LIN {X 0,Y 539.247,Z 614.547,A -85,B 0,C 180,E1 4148.067,E2 4148.067} C_VEL
LIN {X 0,Y 539.704,Z 596.852,A -85,B 0,C 180,E1 4151.322,E2 4151.322} C_VEL
LIN {X 0,Y 540.471,Z 575.476,A -85,B 0,C 180,E1 4153.979,E2 4153.979} C_VEL
LIN {X 0,Y 541.317,Z 550.513,A -85,B 0,C 180,E1 4156.103,E2 4156.103} C_VEL
LIN {X 0,Y 542.051,Z 521.445,A -85,B 0,C 180,E1 4157.733,E2 4157.733} C_VEL
LIN {X 0,Y 542.484,Z 497.198,A -85,B 0,C 180,E1 4158.573,E2 4158.573} C_VEL
LIN {X 0,Y 539.142,Z 489.589,A -85,B 0,C 180,E1 4158.86,E2 4158.86} C_VEL
LIN {X 0,Y 531.289,Z 479.104,A -85,B 0,C 180,E1 4159.277,E2 4159.277} C_VEL
LIN {X 0,Y 530.945,Z 477.682,A -85,B 0,C 180,E1 4159.309,E2 4159.309} C_VEL
LIN {X 0,Y 530.735,Z 476.03,A -85,B 0,C 180,E1 4159.457,E2 4159.457} C_VEL
LIN {X 0,Y 530.499,Z 476.03,A -85,B 0,C 180,E1 4165.344,E2 4165.344} C_VEL
LIN {X 0,Y 530.255,Z 476.03,A -85,B 0,C 180,E1 4171.059,E2 4171.059} C_VEL
LIN {X 0,Y 530.287,Z 476.03,A -85,B 0,C 180,E1 4176.919,E2 4176.919} C_VEL
LIN {X 0,Y 530.344,Z 476.03,A -85,B 0,C 180,E1 4183.243,E2 4183.243} C_VEL
LIN {X 0,Y 530.21,Z 476.03,A -85,B 0,C 180,E1 4188.943,E2 4188.943} C_VEL
LIN {X 0,Y 530.367,Z 476.503,A -85,B 0,C 180,E1 4195.274,E2 4195.274} C_VEL
LIN {X 0,Y 532.518,Z 481.45,A -85,B 0,C 180,E1 4195.82,E2 4195.82} C_VEL
LIN {X 0,Y 542.624,Z 503.518,A -85,B 0,C 180,E1 4196.884,E2 4196.884} C_VEL
LIN {X 0,Y 542.117,Z 551.678,A -85,B 0,C 180,E1 4197.799,E2 4197.799} C_VEL
LIN {X 0,Y 540.712,Z 589.964,A -85,B 0,C 180,E1 4199.149,E2 4199.149} C_VEL
LIN {X 0,Y 538.696,Z 626.732,A -85,B 0,C 180,E1 4201.093,E2 4201.093} C_VEL
LIN {X 0,Y 536.576,Z 662.272,A -85,B 0,C 180,E1 4203.713,E2 4203.713} C_VEL
LIN {X 0,Y 534.555,Z 694.095,A -85,B 0,C 180,E1 4206.848,E2 4206.848} C_VEL
LIN {X 0,Y 532.935,Z 722.17,A -85,B 0,C 180,E1 4210.498,E2 4210.498} C_VEL
LIN {X 0,Y 531.902,Z 745.31,A -85,B 0,C 180,E1 4214.522,E2 4214.522} C_VEL
LIN {X 0,Y 531.296,Z 763.002,A -85,B 0,C 180,E1 4218.819,E2 4218.819} C_VEL
LIN {X 0,Y 531.132,Z 773.548,A -85,B 0,C 180,E1 4222.629,E2 4222.629} C_VEL
LIN {X 0,Y 531.001,Z 779.923,A -85,B 0,C 180,E1 4226.73,E2 4226.73} C_VEL
LIN {X 0,Y 531.003,Z 781.5,A -85,B 0,C 180,E1 4230,E2 4230} C_VEL
LIN {X 0,Y 531.007,Z 779.437,A -85,B 0,C 180,E1 4233.737,E2 4233.737} C_VEL
LIN {X 0,Y 531.193,Z 773.549,A -85,B 0,C 180,E1 4237.369,E2 4237.369} C_VEL
LIN {X 0,Y 531.407,Z 761.9,A -85,B 0,C 180,E1 4241.504,E2 4241.504} C_VEL
LIN {X 0,Y 531.939,Z 744.256,A -85,B 0,C 180,E1 4245.688,E2 4245.688} C_VEL
LIN {X 0,Y 533.035,Z 720.739,A -85,B 0,C 180,E1 4249.713,E2 4249.713} C_VEL
LIN {X 0,Y 534.71,Z 692.275,A -85,B 0,C 180,E1 4253.355,E2 4253.355} C_VEL
LIN {X 0,Y 536.74,Z 659.787,A -85,B 0,C 180,E1 4256.497,E2 4256.497} C_VEL
LIN {X 0,Y 538.885,Z 624.595,A -85,B 0,C 180,E1 4259.036,E2 4259.036} C_VEL
LIN {X 0,Y 540.782,Z 587.023,A -85,B 0,C 180,E1 4260.98,E2 4260.98} C_VEL
LIN {X 0,Y 542.348,Z 549.13,A -85,B 0,C 180,E1 4262.256,E2 4262.256} C_VEL
LIN {X 0,Y 542.002,Z 501.739,A -85,B 0,C 180,E1 4263.186,E2 4263.186} C_VEL
LIN {X 0,Y 532.957,Z 482.108,A -85,B 0,C 180,E1 4264.227,E2 4264.227} C_VEL
LIN {X 0,Y 530.337,Z 476.813,A -85,B 0,C 180,E1 4265.348,E2 4265.348} C_VEL
LIN {X 0,Y 530.278,Z 476.03,A -85,B 0,C 180,E1 4271.05,E2 4271.05} C_VEL
LIN {X 0,Y 530.271,Z 476.03,A -85,B 0,C 180,E1 4276.749,E2 4276.749} C_VEL
LIN {X 0,Y 530.233,Z 476.03,A -85,B 0,C 180,E1 4283.16,E2 4283.16} C_VEL
LIN {X 0,Y 530.371,Z 476.03,A -85,B 0,C 180,E1 4289.084,E2 4289.084} C_VEL
LIN {X 0,Y 530.381,Z 476.03,A -85,B 0,C 180,E1 4294.65,E2 4294.65} C_VEL
LIN {X 0,Y 530.532,Z 476.03,A -85,B 0,C 180,E1 4300.356,E2 4300.356} C_VEL
LIN {X 0,Y 530.613,Z 476.03,A -85,B 0,C 180,E1 4305.976,E2 4305.976} C_VEL
LIN {X 0,Y 530.721,Z 476.03,A -85,B 0,C 180,E1 4311.802,E2 4311.802} C_VEL
LIN {X 0,Y 530.902,Z 476.03,A -85,B 0,C 180,E1 4316.733,E2 4316.733} C_VEL
LIN {X 0,Y 530.989,Z 476.03,A -85,B 0,C 180,E1 4321.636,E2 4321.636} C_VEL
LIN {X 0,Y 530.878,Z 476.03,A -85,B 0,C 180,E1 4326.553,E2 4326.553} C_VEL
LIN {X 0,Y 530.677,Z 476.03,A -85,B 0,C 180,E1 4331.522,E2 4331.522} C_VEL
LIN {X 0,Y 530.569,Z 476.03,A -85,B 0,C 180,E1 4336.583,E2 4336.583} C_VEL
LIN {X 0,Y 530.55,Z 476.03,A -85,B 0,C 180,E1 4341.778,E2 4341.778} C_VEL
LIN {X 0,Y 530.375,Z 476.03,A -85,B 0,C 180,E1 4347.75,E2 4347.75} C_VEL
LIN {X 0,Y 530.316,Z 476.03,A -85,B 0,C 180,E1 4354.108,E2 4354.108} C_VEL
LIN {X 0,Y 530.322,Z 476.03,A -85,B 0,C 180,E1 4359.568,E2 4359.568} C_VEL
LIN {X 0,Y 530.322,Z 476.03,A -85,B 0,C 180,E1 4365.542,E2 4365.542} C_VEL
LIN {X 0,Y 530.274,Z 476.03,A -85,B 0,C 180,E1 4371.085,E2 4371.085} C_VEL
LIN {X 0,Y 530.239,Z 476.03,A -85,B 0,C 180,E1 4377.143,E2 4377.143} C_VEL
LIN {X 0,Y 530.401,Z 476.03,A -85,B 0,C 180,E1 4382.823,E2 4382.823} C_VEL
LIN {X 0,Y 530.547,Z 476.03,A -85,B 0,C 180,E1 4388.223,E2 4388.223} C_VEL
LIN {X 0,Y 530.576,Z 476.22,A -85,B 0,C 180,E1 4393.809,E2 4393.809} C_VEL
LIN {X 0,Y 541.216,Z 505.792,A -85,B 0,C 180,E1 4395.529,E2 4395.529} C_VEL
LIN {X 0,Y 539.385,Z 544.707,A -85,B 0,C 180,E1 4397.332,E2 4397.332} C_VEL
LIN {X 0,Y 537.207,Z 582.328,A -85,B 0,C 180,E1 4399.854,E2 4399.854} C_VEL
LIN {X 0,Y 535.231,Z 613.725,A -85,B 0,C 180,E1 4402.687,E2 4402.687} C_VEL
LIN {X 0,Y 533.459,Z 642.916,A -85,B 0,C 180,E1 4406.135,E2 4406.135} C_VEL
LIN {X 0,Y 532.186,Z 667.585,A -85,B 0,C 180,E1 4410,E2 4410} C_VEL
LIN {X 0,Y 531.51,Z 686.382,A -85,B 0,C 180,E1 4413.974,E2 4413.974} C_VEL
LIN {X 0,Y 531.15,Z 700.214,A -85,B 0,C 180,E1 4418.195,E2 4418.195} C_VEL
LIN {X 0,Y 531.001,Z 708.396,A -85,B 0,C 180,E1 4422.349,E2 4422.349} C_VEL
LIN {X 0,Y 530.857,Z 711.428,A -85,B 0,C 180,E1 4426.572,E2 4426.572} C_VEL
LIN {X 0,Y 530.911,Z 709.233,A -85,B 0,C 180,E1 4430.885,E2 4430.885} C_VEL
LIN {X 0,Y 531.121,Z 702.653,A -85,B 0,C 180,E1 4434.71,E2 4434.71} C_VEL
LIN {X 0,Y 531.447,Z 690.039,A -85,B 0,C 180,E1 4438.969,E2 4438.969} C_VEL
LIN {X 0,Y 531.996,Z 672.502,A -85,B 0,C 180,E1 4442.987,E2 4442.987} C_VEL
LIN {X 0,Y 533.086,Z 649.768,A -85,B 0,C 180,E1 4446.803,E2 4446.803} C_VEL
LIN {X 0,Y 534.693,Z 622.228,A -85,B 0,C 180,E1 4450.316,E2 4450.316} C_VEL
LIN {X 0,Y 536.712,Z 590.06,A -85,B 0,C 180,E1 4453.425,E2 4453.425} C_VEL
LIN {X 0,Y 538.829,Z 554.61,A -85,B 0,C 180,E1 4455.99,E2 4455.99} C_VEL
LIN {X 0,Y 540.802,Z 517.426,A -85,B 0,C 180,E1 4457.916,E2 4457.916} C_VEL
LIN {X 0,Y 540.909,Z 503.739,A -85,B 0,C 180,E1 4458.49,E2 4458.49} C_VEL
LIN {X 0,Y 530.23,Z 476.03,A -85,B 0,C 180,E1 4460.193,E2 4460.193} C_VEL
LIN {X 0,Y 530.366,Z 476.03,A -85,B 0,C 180,E1 4465.885,E2 4465.885} C_VEL
LIN {X 0,Y 530.428,Z 476.03,A -85,B 0,C 180,E1 4470.969,E2 4470.969} C_VEL
LIN {X 0,Y 530.383,Z 476.03,A -85,B 0,C 180,E1 4476.442,E2 4476.442} C_VEL
LIN {X 0,Y 530.49,Z 476.03,A -85,B 0,C 180,E1 4480.472,E2 4480.472} C_VEL
LIN {X 0,Y 534.953,Z 498.482,A -85,B 0,C 180,E1 4481.097,E2 4481.097} C_VEL
LIN {X 0,Y 534.252,Z 528.929,A -85,B 0,C 180,E1 4482.261,E2 4482.261} C_VEL
LIN {X 0,Y 533.467,Z 557.152,A -85,B 0,C 180,E1 4484.039,E2 4484.039} C_VEL
LIN {X 0,Y 532.623,Z 580.694,A -85,B 0,C 180,E1 4486.225,E2 4486.225} C_VEL
LIN {X 0,Y 531.918,Z 601.175,A -85,B 0,C 180,E1 4488.969,E2 4488.969} C_VEL
LIN {X 0,Y 531.468,Z 615.613,A -85,B 0,C 180,E1 4491.809,E2 4491.809} C_VEL
LIN {X 0,Y 531.266,Z 626.066,A -85,B 0,C 180,E1 4495.093,E2 4495.093} C_VEL
LIN {X 0,Y 531.115,Z 631.004,A -85,B 0,C 180,E1 4498.364,E2 4498.364} C_VEL
LIN {X 0,Y 531.116,Z 630.95,A -85,B 0,C 180,E1 4501.631,E2 4501.631} C_VEL
LIN {X 0,Y 531.225,Z 625.96,A -85,B 0,C 180,E1 4504.902,E2 4504.902} C_VEL
LIN {X 0,Y 531.465,Z 615.454,A -85,B 0,C 180,E1 4508.186,E2 4508.186} C_VEL
LIN {X 0,Y 532.021,Z 599.451,A -85,B 0,C 180,E1 4511.268,E2 4511.268} C_VEL
LIN {X 0,Y 532.805,Z 578.439,A -85,B 0,C 180,E1 4513.975,E2 4513.975} C_VEL
LIN {X 0,Y 533.692,Z 553.508,A -85,B 0,C 180,E1 4516.17,E2 4516.17} C_VEL
LIN {X 0,Y 534.446,Z 524.927,A -85,B 0,C 180,E1 4517.834,E2 4517.834} C_VEL
LIN {X 0,Y 534.92,Z 493.957,A -85,B 0,C 180,E1 4518.888,E2 4518.888} C_VEL
LIN {X 0,Y 530.945,Z 477.682,A -85,B 0,C 180,E1 4519.309,E2 4519.309} C_VEL
LIN {X 0,Y 529.475,Z 473.72,A -85,B 0,C 180,E1 4519.704,E2 4519.704} C_VEL
LIN {X 0,Y 526.146,Z 472.639,A -85,B 0,C 180,E1 4520.776,E2 4520.776} C_VEL
LIN {X 0,Y 522.532,Z 476.03,A -85,B 0,C 180,E1 4522.997,E2 4522.997} C_VEL
LIN {X 0,Y 522.452,Z 476.03,A -85,B 0,C 180,E1 4527.621,E2 4527.621} C_VEL
LIN {X 0,Y 522.345,Z 476.03,A -85,B 0,C 180,E1 4533.413,E2 4533.413} C_VEL
LIN {X 0,Y 522.405,Z 476.03,A -85,B 0,C 180,E1 4539.609,E2 4539.609} C_VEL
LIN {X 0,Y 522.398,Z 476.03,A -85,B 0,C 180,E1 4545.923,E2 4545.923} C_VEL
LIN {X 0,Y 522.272,Z 476.03,A -85,B 0,C 180,E1 4551.504,E2 4551.504} C_VEL
LIN {X 0,Y 522.352,Z 476.148,A -85,B 0,C 180,E1 4554.345,E2 4554.345} C_VEL
LIN {X 0,Y 523.947,Z 480.754,A -85,B 0,C 180,E1 4554.74,E2 4554.74} C_VEL
LIN {X 0,Y 527.796,Z 488.345,A -85,B 0,C 180,E1 4555.583,E2 4555.583} C_VEL
LIN {X 0,Y 536.066,Z 506.88,A -85,B 0,C 180,E1 4556.479,E2 4556.479} C_VEL
LIN {X 0,Y 535.382,Z 552.945,A -85,B 0,C 180,E1 4557.382,E2 4557.382} C_VEL
LIN {X 0,Y 533.76,Z 592.103,A -85,B 0,C 180,E1 4558.805,E2 4558.805} C_VEL
LIN {X 0,Y 531.495,Z 629.464,A -85,B 0,C 180,E1 4560.849,E2 4560.849} C_VEL
LIN {X 0,Y 529.142,Z 664.928,A -85,B 0,C 180,E1 4563.556,E2 4563.556} C_VEL
LIN {X 0,Y 526.827,Z 697.28,A -85,B 0,C 180,E1 4566.864,E2 4566.864} C_VEL
LIN {X 0,Y 525.14,Z 724.953,A -85,B 0,C 180,E1 4570.635,E2 4570.635} C_VEL
LIN {X 0,Y 524.066,Z 746.308,A -85,B 0,C 180,E1 4574.499,E2 4574.499} C_VEL
LIN {X 0,Y 523.413,Z 763.04,A -85,B 0,C 180,E1 4578.66,E2 4578.66} C_VEL
LIN {X 0,Y 523.257,Z 773.548,A -85,B 0,C 180,E1 4582.518,E2 4582.518} C_VEL
LIN {X 0,Y 523.117,Z 779.926,A -85,B 0,C 180,E1 4586.681,E2 4586.681} C_VEL
LIN {X 0,Y 523.114,Z 781.5,A -85,B 0,C 180,E1 4590,E2 4590} C_VEL
LIN {X 0,Y 523.173,Z 779.927,A -85,B 0,C 180,E1 4593.318,E2 4593.318} C_VEL
LIN {X 0,Y 523.313,Z 773.549,A -85,B 0,C 180,E1 4597.481,E2 4597.481} C_VEL
LIN {X 0,Y 523.542,Z 761.899,A -85,B 0,C 180,E1 4601.68,E2 4601.68} C_VEL
LIN {X 0,Y 524.109,Z 744.255,A -85,B 0,C 180,E1 4605.929,E2 4605.929} C_VEL
LIN {X 0,Y 525.393,Z 720.741,A -85,B 0,C 180,E1 4610.012,E2 4610.012} C_VEL
LIN {X 0,Y 527.246,Z 692.279,A -85,B 0,C 180,E1 4613.706,E2 4613.706} C_VEL
LIN {X 0,Y 529.499,Z 659.852,A -85,B 0,C 180,E1 4616.882,E2 4616.882} C_VEL
LIN {X 0,Y 531.856,Z 624.968,A -85,B 0,C 180,E1 4619.432,E2 4619.432} C_VEL
LIN {X 0,Y 533.86,Z 588.816,A -85,B 0,C 180,E1 4621.344,E2 4621.344} C_VEL
LIN {X 0,Y 535.619,Z 550.484,A -85,B 0,C 180,E1 4622.675,E2 4622.675} C_VEL
LIN {X 0,Y 535.515,Z 504.687,A -85,B 0,C 180,E1 4623.595,E2 4623.595} C_VEL
LIN {X 0,Y 528.216,Z 489.449,A -85,B 0,C 180,E1 4624.37,E2 4624.37} C_VEL
LIN {X 0,Y 523.102,Z 479.252,A -85,B 0,C 180,E1 4625.869,E2 4625.869} C_VEL
LIN {X 0,Y 522.384,Z 476.03,A -85,B 0,C 180,E1 4626.259,E2 4626.259} C_VEL
LIN {X 0,Y 522.392,Z 476.03,A -85,B 0,C 180,E1 4631.808,E2 4631.808} C_VEL
LIN {X 0,Y 522.295,Z 476.03,A -85,B 0,C 180,E1 4638.19,E2 4638.19} C_VEL
LIN {X 0,Y 522.325,Z 476.03,A -85,B 0,C 180,E1 4644.572,E2 4644.572} C_VEL
LIN {X 0,Y 522.419,Z 476.03,A -85,B 0,C 180,E1 4650.487,E2 4650.487} C_VEL
LIN {X 0,Y 522.489,Z 476.03,A -85,B 0,C 180,E1 4656.069,E2 4656.069} C_VEL
LIN {X 0,Y 522.628,Z 476.03,A -85,B 0,C 180,E1 4661.421,E2 4661.421} C_VEL
LIN {X 0,Y 522.747,Z 476.03,A -85,B 0,C 180,E1 4666.605,E2 4666.605} C_VEL
LIN {X 0,Y 522.803,Z 476.03,A -85,B 0,C 180,E1 4671.677,E2 4671.677} C_VEL
LIN {X 0,Y 523.019,Z 476.03,A -85,B 0,C 180,E1 4676.684,E2 4676.684} C_VEL
LIN {X 0,Y 523.081,Z 476.03,A -85,B 0,C 180,E1 4681.661,E2 4681.661} C_VEL
LIN {X 0,Y 522.95,Z 476.03,A -85,B 0,C 180,E1 4686.653,E2 4686.653} C_VEL
LIN {X 0,Y 522.744,Z 476.03,A -85,B 0,C 180,E1 4691.7,E2 4691.7} C_VEL
LIN {X 0,Y 522.609,Z 476.03,A -85,B 0,C 180,E1 4697.044,E2 4697.044} C_VEL
LIN {X 0,Y 522.616,Z 476.03,A -85,B 0,C 180,E1 4702.126,E2 4702.126} C_VEL
LIN {X 0,Y 522.481,Z 476.03,A -85,B 0,C 180,E1 4707.625,E2 4707.625} C_VEL
LIN {X 0,Y 522.392,Z 476.03,A -85,B 0,C 180,E1 4713.415,E2 4713.415} C_VEL
LIN {X 0,Y 522.418,Z 476.03,A -85,B 0,C 180,E1 4719.615,E2 4719.615} C_VEL
LIN {X 0,Y 522.434,Z 476.03,A -85,B 0,C 180,E1 4725.928,E2 4725.928} C_VEL
LIN {X 0,Y 522.325,Z 476.03,A -85,B 0,C 180,E1 4731.505,E2 4731.505} C_VEL
LIN {X 0,Y 522.35,Z 476.03,A -85,B 0,C 180,E1 4737.203,E2 4737.203} C_VEL
LIN {X 0,Y 522.46,Z 476.03,A -85,B 0,C 180,E1 4742.375,E2 4742.375} C_VEL
LIN {X 0,Y 522.626,Z 476.03,A -85,B 0,C 180,E1 4747.981,E2 4747.981} C_VEL
LIN {X 0,Y 522.696,Z 476.803,A -85,B 0,C 180,E1 4753.259,E2 4753.259} C_VEL
LIN {X 0,Y 534.354,Z 507.589,A -85,B 0,C 180,E1 4755.154,E2 4755.154} C_VEL
LIN {X 0,Y 532.357,Z 545.544,A -85,B 0,C 180,E1 4756.953,E2 4756.953} C_VEL
LIN {X 0,Y 529.992,Z 582.961,A -85,B 0,C 180,E1 4759.507,E2 4759.507} C_VEL
LIN {X 0,Y 527.703,Z 615.542,A -85,B 0,C 180,E1 4762.518,E2 4762.518} C_VEL
LIN {X 0,Y 525.768,Z 644.778,A -85,B 0,C 180,E1 4766.078,E2 4766.078} C_VEL
LIN {X 0,Y 524.34,Z 670.089,A -85,B 0,C 180,E1 4770.207,E2 4770.207} C_VEL
LIN {X 0,Y 523.628,Z 687.734,A -85,B 0,C 180,E1 4774.137,E2 4774.137} C_VEL
LIN {X 0,Y 523.253,Z 700.899,A -85,B 0,C 180,E1 4778.319,E2 4778.319} C_VEL
LIN {X 0,Y 523.093,Z 708.707,A -85,B 0,C 180,E1 4782.539,E2 4782.539} C_VEL
LIN {X 0,Y 522.927,Z 711.481,A -85,B 0,C 180,E1 4786.831,E2 4786.831} C_VEL
LIN {X 0,Y 523.026,Z 708.899,A -85,B 0,C 180,E1 4791.215,E2 4791.215} C_VEL
LIN {X 0,Y 523.253,Z 701.922,A -85,B 0,C 180,E1 4795.145,E2 4795.145} C_VEL
LIN {X 0,Y 523.574,Z 690.879,A -85,B 0,C 180,E1 4798.923,E2 4798.923} C_VEL
LIN {X 0,Y 524.186,Z 673.115,A -85,B 0,C 180,E1 4803.107,E2 4803.107} C_VEL
LIN {X 0,Y 525.368,Z 650.852,A -85,B 0,C 180,E1 4806.945,E2 4806.945} C_VEL
LIN {X 0,Y 527.251,Z 622.144,A -85,B 0,C 180,E1 4810.677,E2 4810.677} C_VEL
LIN {X 0,Y 529.548,Z 589.152,A -85,B 0,C 180,E1 4813.893,E2 4813.893} C_VEL
LIN {X 0,Y 531.773,Z 555.053,A -85,B 0,C 180,E1 4816.384,E2 4816.384} C_VEL
LIN {X 0,Y 533.964,Z 517.89,A -85,B 0,C 180,E1 4818.335,E2 4818.335} C_VEL
LIN {X 0,Y 533.752,Z 505.658,A -85,B 0,C 180,E1 4818.881,E2 4818.881} C_VEL
LIN {X 0,Y 522.34,Z 476.03,A -85,B 0,C 180,E1 4820.756,E2 4820.756} C_VEL
LIN {X 0,Y 522.477,Z 476.03,A -85,B 0,C 180,E1 4827.184,E2 4827.184} C_VEL
LIN {X 0,Y 522.428,Z 476.03,A -85,B 0,C 180,E1 4832.372,E2 4832.372} C_VEL
LIN {X 0,Y 522.501,Z 476.03,A -85,B 0,C 180,E1 4838.019,E2 4838.019} C_VEL
LIN {X 0,Y 522.576,Z 476.03,A -85,B 0,C 180,E1 4840.209,E2 4840.209} C_VEL
LIN {X 0,Y 527.382,Z 499.062,A -85,B 0,C 180,E1 4840.851,E2 4840.851} C_VEL
LIN {X 0,Y 526.676,Z 530.113,A -85,B 0,C 180,E1 4842.051,E2 4842.051} C_VEL
LIN {X 0,Y 525.903,Z 557.692,A -85,B 0,C 180,E1 4843.803,E2 4843.803} C_VEL
LIN {X 0,Y 524.978,Z 581.471,A -85,B 0,C 180,E1 4846.021,E2 4846.021} C_VEL
LIN {X 0,Y 524.285,Z 600.962,A -85,B 0,C 180,E1 4848.615,E2 4848.615} C_VEL
LIN {X 0,Y 523.73,Z 616.718,A -85,B 0,C 180,E1 4851.687,E2 4851.687} C_VEL
LIN {X 0,Y 523.509,Z 627.272,A -85,B 0,C 180,E1 4855.02,E2 4855.02} C_VEL
LIN {X 0,Y 523.341,Z 632.303,A -85,B 0,C 180,E1 4858.34,E2 4858.34} C_VEL
LIN {X 0,Y 523.342,Z 632.302,A -85,B 0,C 180,E1 4861.655,E2 4861.655} C_VEL
LIN {X 0,Y 523.469,Z 627.295,A -85,B 0,C 180,E1 4864.975,E2 4864.975} C_VEL
LIN {X 0,Y 523.761,Z 616.75,A -85,B 0,C 180,E1 4868.308,E2 4868.308} C_VEL
LIN {X 0,Y 524.343,Z 600.908,A -85,B 0,C 180,E1 4871.392,E2 4871.392} C_VEL
LIN {X 0,Y 525.063,Z 581.371,A -85,B 0,C 180,E1 4873.972,E2 4873.972} C_VEL
LIN {X 0,Y 526.047,Z 557.177,A -85,B 0,C 180,E1 4876.187,E2 4876.187} C_VEL
LIN {X 0,Y 526.817,Z 529.535,A -85,B 0,C 180,E1 4877.885,E2 4877.885} C_VEL
LIN {X 0,Y 527.321,Z 499.757,A -85,B 0,C 180,E1 4878.989,E2 4878.989} C_VEL
LIN {X 0,Y 525.63,Z 488.068,A -85,B 0,C 180,E1 4879.303,E2 4879.303} C_VEL
LIN {X 0,Y 522.848,Z 476.03,A -85,B 0,C 180,E1 4879.598,E2 4879.598} C_VEL
LIN {X 0,Y 522.532,Z 476.03,A -85,B 0,C 180,E1 4882.997,E2 4882.997} C_VEL
LIN {X 0,Y 520.003,Z 476.03,A -85,B 0,C 180,E1 4884.405,E2 4884.405} C_VEL
LIN {X 0,Y 514.507,Z 476.03,A -85,B 0,C 180,E1 4886.76,E2 4886.76} C_VEL
LIN {X 0,Y 514.399,Z 476.03,A -85,B 0,C 180,E1 4891.988,E2 4891.988} C_VEL
LIN {X 0,Y 514.428,Z 476.03,A -85,B 0,C 180,E1 4898.17,E2 4898.17} C_VEL
LIN {X 0,Y 514.498,Z 476.03,A -85,B 0,C 180,E1 4902.631,E2 4902.631} C_VEL
LIN {X 0,Y 514.419,Z 476.03,A -85,B 0,C 180,E1 4907.392,E2 4907.392} C_VEL
LIN {X 0,Y 514.4,Z 476.03,A -85,B 0,C 180,E1 4913.853,E2 4913.853} C_VEL
LIN {X 0,Y 517.886,Z 485.516,A -85,B 0,C 180,E1 4914.534,E2 4914.534} C_VEL
LIN {X 0,Y 523.589,Z 495.553,A -85,B 0,C 180,E1 4915.385,E2 4915.385} C_VEL
LIN {X 0,Y 529.466,Z 509.691,A -85,B 0,C 180,E1 4916.049,E2 4916.049} C_VEL
LIN {X 0,Y 528.646,Z 554.89,A -85,B 0,C 180,E1 4916.975,E2 4916.975} C_VEL
LIN {X 0,Y 526.855,Z 593.492,A -85,B 0,C 180,E1 4918.418,E2 4918.418} C_VEL
LIN {X 0,Y 524.414,Z 630.403,A -85,B 0,C 180,E1 4920.482,E2 4920.482} C_VEL
LIN {X 0,Y 521.864,Z 664.934,A -85,B 0,C 180,E1 4923.158,E2 4923.158} C_VEL
LIN {X 0,Y 519.387,Z 697.28,A -85,B 0,C 180,E1 4926.513,E2 4926.513} C_VEL
LIN {X 0,Y 517.459,Z 724.954,A -85,B 0,C 180,E1 4930.336,E2 4930.336} C_VEL
LIN {X 0,Y 516.251,Z 746.309,A -85,B 0,C 180,E1 4934.258,E2 4934.258} C_VEL
LIN {X 0,Y 515.568,Z 761.895,A -85,B 0,C 180,E1 4938.136,E2 4938.136} C_VEL
LIN {X 0,Y 515.356,Z 773.547,A -85,B 0,C 180,E1 4942.402,E2 4942.402} C_VEL
LIN {X 0,Y 515.211,Z 779.929,A -85,B 0,C 180,E1 4946.63,E2 4946.63} C_VEL
LIN {X 0,Y 515.214,Z 781.5,A -85,B 0,C 180,E1 4950,E2 4950} C_VEL
LIN {X 0,Y 515.278,Z 779.929,A -85,B 0,C 180,E1 4953.369,E2 4953.369} C_VEL
LIN {X 0,Y 515.433,Z 773.548,A -85,B 0,C 180,E1 4957.596,E2 4957.596} C_VEL
LIN {X 0,Y 515.664,Z 761.898,A -85,B 0,C 180,E1 4961.861,E2 4961.861} C_VEL
LIN {X 0,Y 516.324,Z 744.255,A -85,B 0,C 180,E1 4966.176,E2 4966.176} C_VEL
LIN {X 0,Y 517.711,Z 720.74,A -85,B 0,C 180,E1 4970.322,E2 4970.322} C_VEL
LIN {X 0,Y 519.777,Z 692.283,A -85,B 0,C 180,E1 4974.068,E2 4974.068} C_VEL
LIN {X 0,Y 522.296,Z 659.85,A -85,B 0,C 180,E1 4977.283,E2 4977.283} C_VEL
LIN {X 0,Y 524.906,Z 624.406,A -85,B 0,C 180,E1 4979.898,E2 4979.898} C_VEL
LIN {X 0,Y 527.077,Z 588.718,A -85,B 0,C 180,E1 4981.798,E2 4981.798} C_VEL
LIN {X 0,Y 528.931,Z 551.593,A -85,B 0,C 180,E1 4983.109,E2 4983.109} C_VEL
LIN {X 0,Y 529.011,Z 507.316,A -85,B 0,C 180,E1 4984.022,E2 4984.022} C_VEL
LIN {X 0,Y 521.991,Z 492.878,A -85,B 0,C 180,E1 4984.867,E2 4984.867} C_VEL
LIN {X 0,Y 515.836,Z 481.711,A -85,B 0,C 180,E1 4986.121,E2 4986.121} C_VEL
LIN {X 0,Y 514.502,Z 476.03,A -85,B 0,C 180,E1 4986.634,E2 4986.634} C_VEL
LIN {X 0,Y 514.461,Z 476.03,A -85,B 0,C 180,E1 4992.635,E2 4992.635} C_VEL
LIN {X 0,Y 514.369,Z 476.03,A -85,B 0,C 180,E1 4997.395,E2 4997.395} C_VEL
LIN {X 0,Y 514.359,Z 476.03,A -85,B 0,C 180,E1 5002.636,E2 5002.636} C_VEL
LIN {X 0,Y 514.541,Z 476.03,A -85,B 0,C 180,E1 5008.58,E2 5008.58} C_VEL
LIN {X 0,Y 514.488,Z 476.03,A -85,B 0,C 180,E1 5013.809,E2 5013.809} C_VEL
LIN {X 0,Y 514.601,Z 476.03,A -85,B 0,C 180,E1 5019.329,E2 5019.329} C_VEL
LIN {X 0,Y 514.787,Z 476.03,A -85,B 0,C 180,E1 5024.654,E2 5024.654} C_VEL
LIN {X 0,Y 514.881,Z 476.03,A -85,B 0,C 180,E1 5029.841,E2 5029.841} C_VEL
LIN {X 0,Y 515.109,Z 476.03,A -85,B 0,C 180,E1 5036.633,E2 5036.633} C_VEL
LIN {X 0,Y 515.105,Z 476.03,A -85,B 0,C 180,E1 5041.98,E2 5041.98} C_VEL
LIN {X 0,Y 515.038,Z 476.03,A -85,B 0,C 180,E1 5046.755,E2 5046.755} C_VEL
LIN {X 0,Y 514.814,Z 476.03,A -85,B 0,C 180,E1 5051.883,E2 5051.883} C_VEL
LIN {X 0,Y 514.713,Z 476.03,A -85,B 0,C 180,E1 5057.109,E2 5057.109} C_VEL
LIN {X 0,Y 514.67,Z 476.03,A -85,B 0,C 180,E1 5062.487,E2 5062.487} C_VEL
LIN {X 0,Y 514.528,Z 476.03,A -85,B 0,C 180,E1 5068.089,E2 5068.089} C_VEL
LIN {X 0,Y 514.421,Z 476.03,A -85,B 0,C 180,E1 5074.5,E2 5074.5} C_VEL
LIN {X 0,Y 514.475,Z 476.03,A -85,B 0,C 180,E1 5080.351,E2 5080.351} C_VEL
LIN {X 0,Y 514.442,Z 476.03,A -85,B 0,C 180,E1 5085.06,E2 5085.06} C_VEL
LIN {X 0,Y 514.482,Z 476.03,A -85,B 0,C 180,E1 5089.922,E2 5089.922} C_VEL
LIN {X 0,Y 514.362,Z 476.03,A -85,B 0,C 180,E1 5095.993,E2 5095.993} C_VEL
LIN {X 0,Y 514.52,Z 476.03,A -85,B 0,C 180,E1 5101.984,E2 5101.984} C_VEL
LIN {X 0,Y 514.659,Z 476.03,A -85,B 0,C 180,E1 5107.514,E2 5107.514} C_VEL
LIN {X 0,Y 514.729,Z 476.03,A -85,B 0,C 180,E1 5112.619,E2 5112.619} C_VEL
LIN {X 0,Y 527.453,Z 510.421,A -85,B 0,C 180,E1 5114.809,E2 5114.809} C_VEL
LIN {X 0,Y 525.258,Z 548.077,A -85,B 0,C 180,E1 5116.667,E2 5116.667} C_VEL
LIN {X 0,Y 522.683,Z 584.879,A -85,B 0,C 180,E1 5119.253,E2 5119.253} C_VEL
LIN {X 0,Y 520.142,Z 617.442,A -85,B 0,C 180,E1 5122.353,E2 5122.353} C_VEL
LIN {X 0,Y 518.128,Z 645.137,A -85,B 0,C 180,E1 5125.811,E2 5125.811} C_VEL
LIN {X 0,Y 516.617,Z 669.282,A -85,B 0,C 180,E1 5129.79,E2 5129.79} C_VEL
LIN {X 0,Y 515.781,Z 687.701,A -85,B 0,C 180,E1 5133.93,E2 5133.93} C_VEL
LIN {X 0,Y 515.425,Z 700.468,A -85,B 0,C 180,E1 5138.021,E2 5138.021} C_VEL
LIN {X 0,Y 515.221,Z 707.932,A -85,B 0,C 180,E1 5141.872,E2 5141.872} C_VEL
LIN {X 0,Y 515.018,Z 711.143,A -85,B 0,C 180,E1 5145.343,E2 5145.343} C_VEL
LIN {X 0,Y 515.026,Z 710.33,A -85,B 0,C 180,E1 5149.824,E2 5149.824} C_VEL
LIN {X 0,Y 515.299,Z 704.083,A -85,B 0,C 180,E1 5154.291,E2 5154.291} C_VEL
LIN {X 0,Y 515.695,Z 692.555,A -85,B 0,C 180,E1 5158.607,E2 5158.607} C_VEL
LIN {X 0,Y 516.323,Z 676.158,A -85,B 0,C 180,E1 5162.725,E2 5162.725} C_VEL
LIN {X 0,Y 517.603,Z 653.973,A -85,B 0,C 180,E1 5166.771,E2 5166.771} C_VEL
LIN {X 0,Y 519.535,Z 625.599,A -85,B 0,C 180,E1 5170.632,E2 5170.632} C_VEL
LIN {X 0,Y 521.893,Z 594.634,A -85,B 0,C 180,E1 5173.818,E2 5173.818} C_VEL
LIN {X 0,Y 524.516,Z 559.071,A -85,B 0,C 180,E1 5176.561,E2 5176.561} C_VEL
LIN {X 0,Y 526.915,Z 521.335,A -85,B 0,C 180,E1 5178.631,E2 5178.631} C_VEL
LIN {X 0,Y 527.1,Z 508.865,A -85,B 0,C 180,E1 5179.194,E2 5179.194} C_VEL
LIN {X 0,Y 514.411,Z 476.03,A -85,B 0,C 180,E1 5181.32,E2 5181.32} C_VEL
LIN {X 0,Y 514.555,Z 476.03,A -85,B 0,C 180,E1 5188.017,E2 5188.017} C_VEL
LIN {X 0,Y 514.488,Z 476.03,A -85,B 0,C 180,E1 5193.803,E2 5193.803} C_VEL
LIN {X 0,Y 514.629,Z 476.03,A -85,B 0,C 180,E1 5199.935,E2 5199.935} C_VEL
LIN {X 0,Y 519.755,Z 499.577,A -85,B 0,C 180,E1 5200.594,E2 5200.594} C_VEL
LIN {X 0,Y 519.156,Z 530.337,A -85,B 0,C 180,E1 5201.786,E2 5201.786} C_VEL
LIN {X 0,Y 518.332,Z 558.215,A -85,B 0,C 180,E1 5203.56,E2 5203.56} C_VEL
LIN {X 0,Y 517.319,Z 582.527,A -85,B 0,C 180,E1 5205.842,E2 5205.842} C_VEL
LIN {X 0,Y 516.561,Z 602.748,A -85,B 0,C 180,E1 5208.58,E2 5208.58} C_VEL
LIN {X 0,Y 515.981,Z 617.823,A -85,B 0,C 180,E1 5211.561,E2 5211.561} C_VEL
LIN {X 0,Y 515.735,Z 628.487,A -85,B 0,C 180,E1 5214.945,E2 5214.945} C_VEL
LIN {X 0,Y 515.556,Z 633.593,A -85,B 0,C 180,E1 5218.315,E2 5218.315} C_VEL
LIN {X 0,Y 515.582,Z 633.645,A -85,B 0,C 180,E1 5221.68,E2 5221.68} C_VEL
LIN {X 0,Y 515.734,Z 628.632,A -85,B 0,C 180,E1 5225.05,E2 5225.05} C_VEL
LIN {X 0,Y 516.061,Z 618.044,A -85,B 0,C 180,E1 5228.432,E2 5228.432} C_VEL
LIN {X 0,Y 516.711,Z 601.594,A -85,B 0,C 180,E1 5231.637,E2 5231.637} C_VEL
LIN {X 0,Y 517.601,Z 580.356,A -85,B 0,C 180,E1 5234.394,E2 5234.394} C_VEL
LIN {X 0,Y 518.575,Z 554.86,A -85,B 0,C 180,E1 5236.644,E2 5236.644} C_VEL
LIN {X 0,Y 519.329,Z 527.001,A -85,B 0,C 180,E1 5238.269,E2 5238.269} C_VEL
LIN {X 0,Y 519.745,Z 496.442,A -85,B 0,C 180,E1 5239.316,E2 5239.316} C_VEL
LIN {X 0,Y 514.907,Z 476.03,A -85,B 0,C 180,E1 5239.88,E2 5239.88} C_VEL
LIN {X 0,Y 514.588,Z 476.03,A -85,B 0,C 180,E1 5246.186,E2 5246.186} C_VEL
LIN {X 0,Y 514.507,Z 476.03,A -85,B 0,C 180,E1 5246.76,E2 5246.76} C_VEL
LIN {X 0,Y 510.554,Z 476.03,A -85,B 0,C 180,E1 5248.662,E2 5248.662} C_VEL
LIN {X 0,Y 506.494,Z 476.03,A -85,B 0,C 180,E1 5250.594,E2 5250.594} C_VEL
LIN {X 0,Y 506.514,Z 476.03,A -85,B 0,C 180,E1 5256.71,E2 5256.71} C_VEL
LIN {X 0,Y 506.509,Z 476.03,A -85,B 0,C 180,E1 5263.428,E2 5263.428} C_VEL
LIN {X 0,Y 506.416,Z 476.03,A -85,B 0,C 180,E1 5268.869,E2 5268.869} C_VEL
LIN {X 0,Y 506.47,Z 476.155,A -85,B 0,C 180,E1 5273.39,E2 5273.39} C_VEL
LIN {X 0,Y 512.056,Z 490.769,A -85,B 0,C 180,E1 5274.434,E2 5274.434} C_VEL
LIN {X 0,Y 519.906,Z 504.139,A -85,B 0,C 180,E1 5275.246,E2 5275.246} C_VEL
LIN {X 0,Y 522.752,Z 510.057,A -85,B 0,C 180,E1 5275.559,E2 5275.559} C_VEL
LIN {X 0,Y 522.001,Z 554.884,A -85,B 0,C 180,E1 5276.5,E2 5276.5} C_VEL
LIN {X 0,Y 520.033,Z 594.038,A -85,B 0,C 180,E1 5277.984,E2 5277.984} C_VEL
LIN {X 0,Y 517.419,Z 630.411,A -85,B 0,C 180,E1 5280.042,E2 5280.042} C_VEL
LIN {X 0,Y 514.538,Z 666.185,A -85,B 0,C 180,E1 5282.863,E2 5282.863} C_VEL
LIN {X 0,Y 511.843,Z 698.28,A -85,B 0,C 180,E1 5286.273,E2 5286.273} C_VEL
LIN {X 0,Y 509.782,Z 724.955,A -85,B 0,C 180,E1 5290.027,E2 5290.027} C_VEL
LIN {X 0,Y 508.427,Z 746.311,A -85,B 0,C 180,E1 5294.01,E2 5294.01} C_VEL
LIN {X 0,Y 507.704,Z 761.895,A -85,B 0,C 180,E1 5297.95,E2 5297.95} C_VEL
LIN {X 0,Y 507.456,Z 773.546,A -85,B 0,C 180,E1 5302.283,E2 5302.283} C_VEL
LIN {X 0,Y 507.306,Z 779.932,A -85,B 0,C 180,E1 5306.578,E2 5306.578} C_VEL
LIN {X 0,Y 507.327,Z 781.5,A -85,B 0,C 180,E1 5310,E2 5310} C_VEL
LIN {X 0,Y 507.371,Z 779.932,A -85,B 0,C 180,E1 5313.421,E2 5313.421} C_VEL
LIN {X 0,Y 507.526,Z 773.547,A -85,B 0,C 180,E1 5317.715,E2 5317.715} C_VEL
LIN {X 0,Y 507.818,Z 761.897,A -85,B 0,C 180,E1 5322.047,E2 5322.047} C_VEL
LIN {X 0,Y 508.55,Z 744.254,A -85,B 0,C 180,E1 5326.43,E2 5326.43} C_VEL
LIN {X 0,Y 510.001,Z 722.172,A -85,B 0,C 180,E1 5330.416,E2 5330.416} C_VEL
LIN {X 0,Y 512.182,Z 694.67,A -85,B 0,C 180,E1 5334.157,E2 5334.157} C_VEL
LIN {X 0,Y 514.879,Z 662.415,A -85,B 0,C 180,E1 5337.472,E2 5337.472} C_VEL
LIN {X 0,Y 517.645,Z 628.347,A -85,B 0,C 180,E1 5340.089,E2 5340.089} C_VEL
LIN {X 0,Y 520.096,Z 592.133,A -85,B 0,C 180,E1 5342.111,E2 5342.111} C_VEL
LIN {X 0,Y 522.19,Z 553.317,A -85,B 0,C 180,E1 5343.538,E2 5343.538} C_VEL
LIN {X 0,Y 522.564,Z 510.181,A -85,B 0,C 180,E1 5344.454,E2 5344.454} C_VEL
LIN {X 0,Y 515.365,Z 496.948,A -85,B 0,C 180,E1 5345.225,E2 5345.225} C_VEL
LIN {X 0,Y 509.297,Z 486.474,A -85,B 0,C 180,E1 5346.148,E2 5346.148} C_VEL
LIN {X 0,Y 506.532,Z 476.03,A -85,B 0,C 180,E1 5347.134,E2 5347.134} C_VEL
LIN {X 0,Y 506.473,Z 476.03,A -85,B 0,C 180,E1 5353.439,E2 5353.439} C_VEL
LIN {X 0,Y 506.388,Z 476.03,A -85,B 0,C 180,E1 5358.874,E2 5358.874} C_VEL
LIN {X 0,Y 506.511,Z 476.03,A -85,B 0,C 180,E1 5365.397,E2 5365.397} C_VEL
LIN {X 0,Y 506.508,Z 476.03,A -85,B 0,C 180,E1 5371.431,E2 5371.431} C_VEL
LIN {X 0,Y 506.653,Z 476.03,A -85,B 0,C 180,E1 5377.883,E2 5377.883} C_VEL
LIN {X 0,Y 506.856,Z 476.03,A -85,B 0,C 180,E1 5382.925,E2 5382.925} C_VEL
LIN {X 0,Y 506.865,Z 476.03,A -85,B 0,C 180,E1 5387.934,E2 5387.934} C_VEL
LIN {X 0,Y 506.964,Z 476.03,A -85,B 0,C 180,E1 5393.142,E2 5393.142} C_VEL
LIN {X 0,Y 507.082,Z 476.03,A -85,B 0,C 180,E1 5398.292,E2 5398.292} C_VEL
LIN {X 0,Y 507.072,Z 476.03,A -85,B 0,C 180,E1 5403.426,E2 5403.426} C_VEL
LIN {X 0,Y 506.914,Z 476.03,A -85,B 0,C 180,E1 5408.591,E2 5408.591} C_VEL
LIN {X 0,Y 506.834,Z 476.03,A -85,B 0,C 180,E1 5413.829,E2 5413.829} C_VEL
LIN {X 0,Y 506.753,Z 476.03,A -85,B 0,C 180,E1 5419.189,E2 5419.189} C_VEL
LIN {X 0,Y 506.702,Z 476.03,A -85,B 0,C 180,E1 5424.731,E2 5424.731} C_VEL
LIN {X 0,Y 506.537,Z 476.03,A -85,B 0,C 180,E1 5430.542,E2 5430.542} C_VEL
LIN {X 0,Y 506.561,Z 476.03,A -85,B 0,C 180,E1 5436.713,E2 5436.713} C_VEL
LIN {X 0,Y 506.46,Z 476.03,A -85,B 0,C 180,E1 5443.441,E2 5443.441} C_VEL
LIN {X 0,Y 506.491,Z 476.03,A -85,B 0,C 180,E1 5448.878,E2 5448.878} C_VEL
LIN {X 0,Y 506.453,Z 476.03,A -85,B 0,C 180,E1 5455.387,E2 5455.387} C_VEL
LIN {X 0,Y 506.536,Z 476.03,A -85,B 0,C 180,E1 5461.428,E2 5461.428} C_VEL
LIN {X 0,Y 506.75,Z 476.03,A -85,B 0,C 180,E1 5467.854,E2 5467.854} C_VEL
LIN {X 0,Y 506.856,Z 476.047,A -85,B 0,C 180,E1 5472.057,E2 5472.057} C_VEL
LIN {X 0,Y 520.632,Z 512.413,A -85,B 0,C 180,E1 5474.423,E2 5474.423} C_VEL
LIN {X 0,Y 518.256,Z 548.878,A -85,B 0,C 180,E1 5476.269,E2 5476.269} C_VEL
LIN {X 0,Y 515.452,Z 585.529,A -85,B 0,C 180,E1 5478.886,E2 5478.886} C_VEL
LIN {X 0,Y 512.574,Z 619.574,A -85,B 0,C 180,E1 5482.209,E2 5482.209} C_VEL
LIN {X 0,Y 510.421,Z 646.9,A -85,B 0,C 180,E1 5485.747,E2 5485.747} C_VEL
LIN {X 0,Y 508.808,Z 670.623,A -85,B 0,C 180,E1 5489.787,E2 5489.787} C_VEL
LIN {X 0,Y 507.898,Z 688.669,A -85,B 0,C 180,E1 5493.992,E2 5493.992} C_VEL
LIN {X 0,Y 507.506,Z 701.123,A -85,B 0,C 180,E1 5498.147,E2 5498.147} C_VEL
LIN {X 0,Y 507.299,Z 708.298,A -85,B 0,C 180,E1 5502.06,E2 5502.06} C_VEL
LIN {X 0,Y 507.088,Z 711.213,A -85,B 0,C 180,E1 5505.589,E2 5505.589} C_VEL
LIN {X 0,Y 507.123,Z 710.807,A -85,B 0,C 180,E1 5509.174,E2 5509.174} C_VEL
LIN {X 0,Y 507.374,Z 705.306,A -85,B 0,C 180,E1 5513.758,E2 5513.758} C_VEL
LIN {X 0,Y 507.699,Z 694.981,A -85,B 0,C 180,E1 5518.016,E2 5518.016} C_VEL
LIN {X 0,Y 508.453,Z 678.689,A -85,B 0,C 180,E1 5522.413,E2 5522.413} C_VEL
LIN {X 0,Y 509.67,Z 657.748,A -85,B 0,C 180,E1 5526.453,E2 5526.453} C_VEL
LIN {X 0,Y 511.668,Z 631.034,A -85,B 0,C 180,E1 5530.336,E2 5530.336} C_VEL
LIN {X 0,Y 514.403,Z 598.192,A -85,B 0,C 180,E1 5533.905,E2 5533.905} C_VEL
LIN {X 0,Y 517.273,Z 562.305,A -85,B 0,C 180,E1 5536.779,E2 5536.779} C_VEL
LIN {X 0,Y 519.832,Z 525.802,A -85,B 0,C 180,E1 5538.886,E2 5538.886} C_VEL
LIN {X 0,Y 520.147,Z 511.123,A -85,B 0,C 180,E1 5539.579,E2 5539.579} C_VEL
LIN {X 0,Y 506.454,Z 476.03,A -85,B 0,C 180,E1 5541.949,E2 5541.949} C_VEL
LIN {X 0,Y 506.562,Z 476.03,A -85,B 0,C 180,E1 5547.451,E2 5547.451} C_VEL
LIN {X 0,Y 506.581,Z 476.03,A -85,B 0,C 180,E1 5553.724,E2 5553.724} C_VEL
LIN {X 0,Y 506.774,Z 476.683,A -85,B 0,C 180,E1 5559.661,E2 5559.661} C_VEL
LIN {X 0,Y 512.233,Z 500.492,A -85,B 0,C 180,E1 5560.346,E2 5560.346} C_VEL
LIN {X 0,Y 511.605,Z 531.165,A -85,B 0,C 180,E1 5561.546,E2 5561.546} C_VEL
LIN {X 0,Y 510.757,Z 558.736,A -85,B 0,C 180,E1 5563.309,E2 5563.309} C_VEL
LIN {X 0,Y 509.641,Z 584.042,A -85,B 0,C 180,E1 5565.712,E2 5565.712} C_VEL
LIN {X 0,Y 508.819,Z 604.584,A -85,B 0,C 180,E1 5568.553,E2 5568.553} C_VEL
LIN {X 0,Y 508.157,Z 620.609,A -85,B 0,C 180,E1 5571.861,E2 5571.861} C_VEL
LIN {X 0,Y 507.976,Z 629.699,A -85,B 0,C 180,E1 5574.867,E2 5574.867} C_VEL
LIN {X 0,Y 507.783,Z 634.886,A -85,B 0,C 180,E1 5578.289,E2 5578.289} C_VEL
LIN {X 0,Y 507.808,Z 634.986,A -85,B 0,C 180,E1 5581.706,E2 5581.706} C_VEL
LIN {X 0,Y 507.976,Z 629.978,A -85,B 0,C 180,E1 5585.127,E2 5585.127} C_VEL
LIN {X 0,Y 508.354,Z 619.335,A -85,B 0,C 180,E1 5588.561,E2 5588.561} C_VEL
LIN {X 0,Y 509.033,Z 603.761,A -85,B 0,C 180,E1 5591.656,E2 5591.656} C_VEL
LIN {X 0,Y 509.834,Z 584.167,A -85,B 0,C 180,E1 5594.304,E2 5594.304} C_VEL
LIN {X 0,Y 510.878,Z 559.905,A -85,B 0,C 180,E1 5596.57,E2 5596.57} C_VEL
LIN {X 0,Y 511.662,Z 532.136,A -85,B 0,C 180,E1 5598.307,E2 5598.307} C_VEL
LIN {X 0,Y 512.169,Z 501.597,A -85,B 0,C 180,E1 5599.445,E2 5599.445} C_VEL
LIN {X 0,Y 508.728,Z 483.598,A -85,B 0,C 180,E1 5599.921,E2 5599.921} C_VEL
LIN {X 0,Y 506.974,Z 476.03,A -85,B 0,C 180,E1 5600.145,E2 5600.145} C_VEL
LIN {X 0,Y 506.612,Z 476.03,A -85,B 0,C 180,E1 5606.741,E2 5606.741} C_VEL
LIN {X 0,Y 506.494,Z 476.03,A -85,B 0,C 180,E1 5610.594,E2 5610.594} C_VEL
LIN {X 0,Y 502.368,Z 476.03,A -85,B 0,C 180,E1 5612.532,E2 5612.532} C_VEL
LIN {X 0,Y 498.503,Z 476.03,A -85,B 0,C 180,E1 5614.501,E2 5614.501} C_VEL
LIN {X 0,Y 498.533,Z 476.03,A -85,B 0,C 180,E1 5620.598,E2 5620.598} C_VEL
LIN {X 0,Y 498.553,Z 476.03,A -85,B 0,C 180,E1 5626.785,E2 5626.785} C_VEL
LIN {X 0,Y 498.513,Z 476.03,A -85,B 0,C 180,E1 5632.892,E2 5632.892} C_VEL
LIN {X 0,Y 503.893,Z 491.226,A -85,B 0,C 180,E1 5633.809,E2 5633.809} C_VEL
LIN {X 0,Y 513.82,Z 507.75,A -85,B 0,C 180,E1 5634.848,E2 5634.848} C_VEL
LIN {X 0,Y 516.359,Z 513.608,A -85,B 0,C 180,E1 5635.133,E2 5635.133} C_VEL
LIN {X 0,Y 515.332,Z 556.576,A -85,B 0,C 180,E1 5636.065,E2 5636.065} C_VEL
LIN {X 0,Y 513.179,Z 595.58,A -85,B 0,C 180,E1 5637.588,E2 5637.588} C_VEL
LIN {X 0,Y 510.308,Z 632.106,A -85,B 0,C 180,E1 5639.708,E2 5639.708} C_VEL
LIN {X 0,Y 507.218,Z 667.388,A -85,B 0,C 180,E1 5642.56,E2 5642.56} C_VEL
LIN {X 0,Y 504.427,Z 698.413,A -85,B 0,C 180,E1 5645.92,E2 5645.92} C_VEL
LIN {X 0,Y 502.089,Z 725.734,A -85,B 0,C 180,E1 5649.841,E2 5649.841} C_VEL
LIN {X 0,Y 500.645,Z 746.312,A -85,B 0,C 180,E1 5653.754,E2 5653.754} C_VEL
LIN {X 0,Y 499.851,Z 761.894,A -85,B 0,C 180,E1 5657.758,E2 5657.758} C_VEL
LIN {X 0,Y 499.571,Z 773.545,A -85,B 0,C 180,E1 5662.161,E2 5662.161} C_VEL
LIN {X 0,Y 499.401,Z 779.935,A -85,B 0,C 180,E1 5666.523,E2 5666.523} C_VEL
LIN {X 0,Y 499.44,Z 781.5,A -85,B 0,C 180,E1 5670,E2 5670} C_VEL
LIN {X 0,Y 499.463,Z 779.935,A -85,B 0,C 180,E1 5673.476,E2 5673.476} C_VEL
LIN {X 0,Y 499.63,Z 773.546,A -85,B 0,C 180,E1 5677.838,E2 5677.838} C_VEL
LIN {X 0,Y 499.957,Z 761.896,A -85,B 0,C 180,E1 5682.239,E2 5682.239} C_VEL
LIN {X 0,Y 500.816,Z 744.253,A -85,B 0,C 180,E1 5686.691,E2 5686.691} C_VEL
LIN {X 0,Y 502.478,Z 720.956,A -85,B 0,C 180,E1 5690.932,E2 5690.932} C_VEL
LIN {X 0,Y 504.982,Z 692.291,A -85,B 0,C 180,E1 5694.82,E2 5694.82} C_VEL
LIN {X 0,Y 507.956,Z 659.844,A -85,B 0,C 180,E1 5698.121,E2 5698.121} C_VEL
LIN {X 0,Y 510.957,Z 624.879,A -85,B 0,C 180,E1 5700.768,E2 5700.768} C_VEL
LIN {X 0,Y 513.596,Z 588.614,A -85,B 0,C 180,E1 5702.74,E2 5702.74} C_VEL
LIN {X 0,Y 515.731,Z 551.215,A -85,B 0,C 180,E1 5704.081,E2 5704.081} C_VEL
LIN {X 0,Y 515.875,Z 512.391,A -85,B 0,C 180,E1 5704.928,E2 5704.928} C_VEL
LIN {X 0,Y 509.679,Z 501.657,A -85,B 0,C 180,E1 5705.597,E2 5705.597} C_VEL
LIN {X 0,Y 501.356,Z 486.802,A -85,B 0,C 180,E1 5706.584,E2 5706.584} C_VEL
LIN {X 0,Y 498.654,Z 476.03,A -85,B 0,C 180,E1 5707.629,E2 5707.629} C_VEL
LIN {X 0,Y 498.548,Z 476.03,A -85,B 0,C 180,E1 5714.308,E2 5714.308} C_VEL
LIN {X 0,Y 498.435,Z 476.03,A -85,B 0,C 180,E1 5720.37,E2 5720.37} C_VEL
LIN {X 0,Y 498.632,Z 476.03,A -85,B 0,C 180,E1 5726.873,E2 5726.873} C_VEL
LIN {X 0,Y 498.598,Z 476.03,A -85,B 0,C 180,E1 5732.907,E2 5732.907} C_VEL
LIN {X 0,Y 498.754,Z 476.03,A -85,B 0,C 180,E1 5738.64,E2 5738.64} C_VEL
LIN {X 0,Y 498.936,Z 476.03,A -85,B 0,C 180,E1 5744.154,E2 5744.154} C_VEL
LIN {X 0,Y 499.024,Z 476.03,A -85,B 0,C 180,E1 5749.514,E2 5749.514} C_VEL
LIN {X 0,Y 499.158,Z 476.03,A -85,B 0,C 180,E1 5754.782,E2 5754.782} C_VEL
LIN {X 0,Y 499.293,Z 476.03,A -85,B 0,C 180,E1 5760.003,E2 5760.003} C_VEL
LIN {X 0,Y 499.196,Z 476.03,A -85,B 0,C 180,E1 5765.223,E2 5765.223} C_VEL
LIN {X 0,Y 499.037,Z 476.03,A -85,B 0,C 180,E1 5770.491,E2 5770.491} C_VEL
LIN {X 0,Y 498.905,Z 476.03,A -85,B 0,C 180,E1 5775.853,E2 5775.853} C_VEL
LIN {X 0,Y 498.833,Z 476.03,A -85,B 0,C 180,E1 5781.362,E2 5781.362} C_VEL
LIN {X 0,Y 498.679,Z 476.03,A -85,B 0,C 180,E1 5787.094,E2 5787.094} C_VEL
LIN {X 0,Y 498.565,Z 476.03,A -85,B 0,C 180,E1 5793.138,E2 5793.138} C_VEL
LIN {X 0,Y 498.536,Z 476.03,A -85,B 0,C 180,E1 5799.628,E2 5799.628} C_VEL
LIN {X 0,Y 498.575,Z 476.03,A -85,B 0,C 180,E1 5805.695,E2 5805.695} C_VEL
LIN {X 0,Y 498.504,Z 476.03,A -85,B 0,C 180,E1 5812.157,E2 5812.157} C_VEL
LIN {X 0,Y 498.499,Z 476.03,A -85,B 0,C 180,E1 5818.26,E2 5818.26} C_VEL
LIN {X 0,Y 498.661,Z 476.03,A -85,B 0,C 180,E1 5822.906,E2 5822.906} C_VEL
LIN {X 0,Y 498.847,Z 476.03,A -85,B 0,C 180,E1 5828.64,E2 5828.64} C_VEL
LIN {X 0,Y 498.946,Z 476.313,A -85,B 0,C 180,E1 5831.453,E2 5831.453} C_VEL
LIN {X 0,Y 513.526,Z 513.704,A -85,B 0,C 180,E1 5833.974,E2 5833.974} C_VEL
LIN {X 0,Y 511.161,Z 551.351,A -85,B 0,C 180,E1 5835.965,E2 5835.965} C_VEL
LIN {X 0,Y 508.275,Z 586.161,A -85,B 0,C 180,E1 5838.509,E2 5838.509} C_VEL
LIN {X 0,Y 505.102,Z 620.691,A -85,B 0,C 180,E1 5841.947,E2 5841.947} C_VEL
LIN {X 0,Y 502.681,Z 648.671,A -85,B 0,C 180,E1 5845.682,E2 5845.682} C_VEL
LIN {X 0,Y 501.008,Z 671.943,A -85,B 0,C 180,E1 5849.784,E2 5849.784} C_VEL
LIN {X 0,Y 500.05,Z 689.103,A -85,B 0,C 180,E1 5853.907,E2 5853.907} C_VEL
LIN {X 0,Y 499.66,Z 700.725,A -85,B 0,C 180,E1 5857.838,E2 5857.838} C_VEL
LIN {X 0,Y 499.361,Z 708.61,A -85,B 0,C 180,E1 5862.254,E2 5862.254} C_VEL
LIN {X 0,Y 499.169,Z 711.274,A -85,B 0,C 180,E1 5865.843,E2 5865.843} C_VEL
LIN {X 0,Y 499.191,Z 710.329,A -85,B 0,C 180,E1 5869.906,E2 5869.906} C_VEL
LIN {X 0,Y 499.479,Z 705.247,A -85,B 0,C 180,E1 5873.9,E2 5873.9} C_VEL
LIN {X 0,Y 499.839,Z 695.023,A -85,B 0,C 180,E1 5878.179,E2 5878.179} C_VEL
LIN {X 0,Y 500.649,Z 678.338,A -85,B 0,C 180,E1 5882.742,E2 5882.742} C_VEL
LIN {X 0,Y 502.177,Z 655.83,A -85,B 0,C 180,E1 5887.087,E2 5887.087} C_VEL
LIN {X 0,Y 504.35,Z 629.417,A -85,B 0,C 180,E1 5890.901,E2 5890.901} C_VEL
LIN {X 0,Y 507.242,Z 597.905,A -85,B 0,C 180,E1 5894.345,E2 5894.345} C_VEL
LIN {X 0,Y 510.357,Z 561.528,A -85,B 0,C 180,E1 5897.284,E2 5897.284} C_VEL
LIN {X 0,Y 513.11,Z 525.364,A -85,B 0,C 180,E1 5899.377,E2 5899.377} C_VEL
LIN {X 0,Y 513.467,Z 514.192,A -85,B 0,C 180,E1 5899.92,E2 5899.92} C_VEL
LIN {X 0,Y 499.228,Z 479.227,A -85,B 0,C 180,E1 5902.322,E2 5902.322} C_VEL
LIN {X 0,Y 498.551,Z 476.03,A -85,B 0,C 180,E1 5902.502,E2 5902.502} C_VEL
LIN {X 0,Y 498.642,Z 476.03,A -85,B 0,C 180,E1 5908.922,E2 5908.922} C_VEL
LIN {X 0,Y 498.682,Z 476.03,A -85,B 0,C 180,E1 5915.627,E2 5915.627} C_VEL
LIN {X 0,Y 498.783,Z 476.03,A -85,B 0,C 180,E1 5919.315,E2 5919.315} C_VEL
LIN {X 0,Y 504.826,Z 502.983,A -85,B 0,C 180,E1 5920.144,E2 5920.144} C_VEL
LIN {X 0,Y 504.024,Z 533.407,A -85,B 0,C 180,E1 5921.374,E2 5921.374} C_VEL
LIN {X 0,Y 503.046,Z 561.966,A -85,B 0,C 180,E1 5923.271,E2 5923.271} C_VEL
LIN {X 0,Y 501.932,Z 586.515,A -85,B 0,C 180,E1 5925.69,E2 5925.69} C_VEL
LIN {X 0,Y 501.11,Z 605.797,A -85,B 0,C 180,E1 5928.418,E2 5928.418} C_VEL
LIN {X 0,Y 500.425,Z 621.709,A -85,B 0,C 180,E1 5931.735,E2 5931.735} C_VEL
LIN {X 0,Y 500.215,Z 630.91,A -85,B 0,C 180,E1 5934.788,E2 5934.788} C_VEL
LIN {X 0,Y 499.994,Z 636.184,A -85,B 0,C 180,E1 5938.262,E2 5938.262} C_VEL
LIN {X 0,Y 500.034,Z 636.326,A -85,B 0,C 180,E1 5941.732,E2 5941.732} C_VEL
LIN {X 0,Y 500.246,Z 631.318,A -85,B 0,C 180,E1 5945.207,E2 5945.207} C_VEL
LIN {X 0,Y 500.644,Z 620.619,A -85,B 0,C 180,E1 5948.694,E2 5948.694} C_VEL
LIN {X 0,Y 501.405,Z 604.403,A -85,B 0,C 180,E1 5951.918,E2 5951.918} C_VEL
LIN {X 0,Y 502.347,Z 583.592,A -85,B 0,C 180,E1 5954.693,E2 5954.693} C_VEL
LIN {X 0,Y 503.383,Z 559.055,A -85,B 0,C 180,E1 5956.937,E2 5956.937} C_VEL
LIN {X 0,Y 504.161,Z 531.408,A -85,B 0,C 180,E1 5958.623,E2 5958.623} C_VEL
LIN {X 0,Y 504.617,Z 501.695,A -85,B 0,C 180,E1 5959.703,E2 5959.703} C_VEL
LIN {X 0,Y 499.021,Z 476.03,A -85,B 0,C 180,E1 5960.419,E2 5960.419} C_VEL
LIN {X 0,Y 498.656,Z 476.03,A -85,B 0,C 180,E1 5967.089,E2 5967.089} C_VEL
LIN {X 0,Y 498.519,Z 476.03,A -85,B 0,C 180,E1 5973.135,E2 5973.135} C_VEL
LIN {X 0,Y 498.503,Z 476.03,A -85,B 0,C 180,E1 5974.501,E2 5974.501} C_VEL
LIN {X 0,Y 496.052,Z 476.03,A -85,B 0,C 180,E1 5975.983,E2 5975.983} C_VEL
LIN {X 0,Y 490.674,Z 476.03,A -85,B 0,C 180,E1 5978.206,E2 5978.206} C_VEL
LIN {X 0,Y 490.573,Z 476.03,A -85,B 0,C 180,E1 5978.463,E2 5978.463} C_VEL
LIN {X 0,Y 490.651,Z 476.03,A -85,B 0,C 180,E1 5984.784,E2 5984.784} C_VEL
LIN {X 0,Y 490.537,Z 476.03,A -85,B 0,C 180,E1 5990.494,E2 5990.494} C_VEL
LIN {X 0,Y 490.618,Z 476.694,A -85,B 0,C 180,E1 5992.427,E2 5992.427} C_VEL
LIN {X 0,Y 501.071,Z 500.382,A -85,B 0,C 180,E1 5993.739,E2 5993.739} C_VEL
LIN {X 0,Y 508.998,Z 514.099,A -85,B 0,C 180,E1 5994.589,E2 5994.589} C_VEL
LIN {X 0,Y 509.717,Z 527.501,A -85,B 0,C 180,E1 5994.889,E2 5994.889} C_VEL
LIN {X 0,Y 507.978,Z 569.382,A -85,B 0,C 180,E1 5996.009,E2 5996.009} C_VEL
LIN {X 0,Y 505.631,Z 605.978,A -85,B 0,C 180,E1 5997.638,E2 5997.638} C_VEL
LIN {X 0,Y 502.511,Z 641.607,A -85,B 0,C 180,E1 5999.938,E2 5999.938} C_VEL
LIN {X 0,Y 499.242,Z 675.567,A -85,B 0,C 180,E1 6002.94,E2 6002.94} C_VEL
LIN {X 0,Y 496.303,Z 705.697,A -85,B 0,C 180,E1 6006.491,E2 6006.491} C_VEL
LIN {X 0,Y 494.099,Z 731.541,A -85,B 0,C 180,E1 6010.531,E2 6010.531} C_VEL
LIN {X 0,Y 492.649,Z 752.43,A -85,B 0,C 180,E1 6014.938,E2 6014.938} C_VEL
LIN {X 0,Y 491.92,Z 767.224,A -85,B 0,C 180,E1 6019.357,E2 6019.357} C_VEL
LIN {X 0,Y 491.629,Z 776.708,A -85,B 0,C 180,E1 6023.812,E2 6023.812} C_VEL
LIN {X 0,Y 491.552,Z 781.109,A -85,B 0,C 180,E1 6028.235,E2 6028.235} C_VEL
LIN {X 0,Y 491.65,Z 781.109,A -85,B 0,C 180,E1 6031.764,E2 6031.764} C_VEL
LIN {X 0,Y 491.613,Z 776.709,A -85,B 0,C 180,E1 6036.188,E2 6036.188} C_VEL
LIN {X 0,Y 491.938,Z 767.227,A -85,B 0,C 180,E1 6040.642,E2 6040.642} C_VEL
LIN {X 0,Y 492.599,Z 752.529,A -85,B 0,C 180,E1 6045.039,E2 6045.039} C_VEL
LIN {X 0,Y 494.134,Z 731.684,A -85,B 0,C 180,E1 6049.441,E2 6049.441} C_VEL
LIN {X 0,Y 496.337,Z 705.642,A -85,B 0,C 180,E1 6053.515,E2 6053.515} C_VEL
LIN {X 0,Y 499.23,Z 675.573,A -85,B 0,C 180,E1 6057.06,E2 6057.06} C_VEL
LIN {X 0,Y 502.504,Z 641.616,A -85,B 0,C 180,E1 6060.062,E2 6060.062} C_VEL
LIN {X 0,Y 505.536,Z 604.883,A -85,B 0,C 180,E1 6062.436,E2 6062.436} C_VEL
LIN {X 0,Y 508.12,Z 566.481,A -85,B 0,C 180,E1 6064.1,E2 6064.1} C_VEL
LIN {X 0,Y 510.023,Z 522.909,A -85,B 0,C 180,E1 6065.2,E2 6065.2} C_VEL
LIN {X 0,Y 509.081,Z 514.47,A -85,B 0,C 180,E1 6065.428,E2 6065.428} C_VEL
LIN {X 0,Y 494.968,Z 489.647,A -85,B 0,C 180,E1 6067.038,E2 6067.038} C_VEL
LIN {X 0,Y 491.515,Z 479.409,A -85,B 0,C 180,E1 6067.736,E2 6067.736} C_VEL
LIN {X 0,Y 490.68,Z 476.03,A -85,B 0,C 180,E1 6068.108,E2 6068.108} C_VEL
LIN {X 0,Y 490.664,Z 476.03,A -85,B 0,C 180,E1 6072.756,E2 6072.756} C_VEL
LIN {X 0,Y 490.563,Z 476.03,A -85,B 0,C 180,E1 6077.796,E2 6077.796} C_VEL
LIN {X 0,Y 490.579,Z 476.03,A -85,B 0,C 180,E1 6084.103,E2 6084.103} C_VEL
LIN {X 0,Y 490.653,Z 476.03,A -85,B 0,C 180,E1 6090.418,E2 6090.418} C_VEL
LIN {X 0,Y 490.77,Z 476.03,A -85,B 0,C 180,E1 6096.359,E2 6096.359} C_VEL
LIN {X 0,Y 490.957,Z 476.03,A -85,B 0,C 180,E1 6102.948,E2 6102.948} C_VEL
LIN {X 0,Y 491.107,Z 476.03,A -85,B 0,C 180,E1 6109.343,E2 6109.343} C_VEL
LIN {X 0,Y 491.242,Z 476.03,A -85,B 0,C 180,E1 6114.698,E2 6114.698} C_VEL
LIN {X 0,Y 491.392,Z 476.03,A -85,B 0,C 180,E1 6120.003,E2 6120.003} C_VEL
LIN {X 0,Y 491.285,Z 476.03,A -85,B 0,C 180,E1 6125.307,E2 6125.307} C_VEL
LIN {X 0,Y 491.119,Z 476.03,A -85,B 0,C 180,E1 6130.662,E2 6130.662} C_VEL
LIN {X 0,Y 490.943,Z 476.03,A -85,B 0,C 180,E1 6137.047,E2 6137.047} C_VEL
LIN {X 0,Y 490.871,Z 476.03,A -85,B 0,C 180,E1 6143.641,E2 6143.641} C_VEL
LIN {X 0,Y 490.639,Z 476.03,A -85,B 0,C 180,E1 6150.222,E2 6150.222} C_VEL
LIN {X 0,Y 490.607,Z 476.03,A -85,B 0,C 180,E1 6156.639,E2 6156.639} C_VEL
LIN {X 0,Y 490.625,Z 476.03,A -85,B 0,C 180,E1 6162.761,E2 6162.761} C_VEL
LIN {X 0,Y 490.683,Z 476.03,A -85,B 0,C 180,E1 6167.78,E2 6167.78} C_VEL
LIN {X 0,Y 490.558,Z 476.03,A -85,B 0,C 180,E1 6174.096,E2 6174.096} C_VEL
LIN {X 0,Y 490.626,Z 476.03,A -85,B 0,C 180,E1 6180.411,E2 6180.411} C_VEL
LIN {X 0,Y 490.858,Z 476.03,A -85,B 0,C 180,E1 6186.359,E2 6186.359} C_VEL
LIN {X 0,Y 490.996,Z 476.117,A -85,B 0,C 180,E1 6190.808,E2 6190.808} C_VEL
LIN {X 0,Y 505.654,Z 513.224,A -85,B 0,C 180,E1 6193.37,E2 6193.37} C_VEL
LIN {X 0,Y 506.734,Z 520.712,A -85,B 0,C 180,E1 6193.827,E2 6193.827} C_VEL
LIN {X 0,Y 503.714,Z 558.82,A -85,B 0,C 180,E1 6195.975,E2 6195.975} C_VEL
LIN {X 0,Y 500.304,Z 595.06,A -85,B 0,C 180,E1 6198.876,E2 6198.876} C_VEL
LIN {X 0,Y 497.273,Z 625.339,A -85,B 0,C 180,E1 6202.116,E2 6202.116} C_VEL
LIN {X 0,Y 494.709,Z 653.236,A -85,B 0,C 180,E1 6206.052,E2 6206.052} C_VEL
LIN {X 0,Y 492.934,Z 676.25,A -85,B 0,C 180,E1 6210.44,E2 6210.44} C_VEL
LIN {X 0,Y 492.093,Z 691.568,A -85,B 0,C 180,E1 6214.412,E2 6214.412} C_VEL
LIN {X 0,Y 491.651,Z 703.23,A -85,B 0,C 180,E1 6218.858,E2 6218.858} C_VEL
LIN {X 0,Y 491.442,Z 708.921,A -85,B 0,C 180,E1 6222.455,E2 6222.455} C_VEL
LIN {X 0,Y 491.207,Z 711.472,A -85,B 0,C 180,E1 6227.151,E2 6227.151} C_VEL
LIN {X 0,Y 491.4,Z 708.641,A -85,B 0,C 180,E1 6231.7,E2 6231.7} C_VEL
LIN {X 0,Y 491.72,Z 700.896,A -85,B 0,C 180,E1 6236.151,E2 6236.151} C_VEL
LIN {X 0,Y 492.33,Z 687.872,A -85,B 0,C 180,E1 6240.56,E2 6240.56} C_VEL
LIN {X 0,Y 493.443,Z 669.075,A -85,B 0,C 180,E1 6244.991,E2 6244.991} C_VEL
LIN {X 0,Y 495.565,Z 644.259,A -85,B 0,C 180,E1 6249.249,E2 6249.249} C_VEL
LIN {X 0,Y 498.352,Z 614.35,A -85,B 0,C 180,E1 6253.073,E2 6253.073} C_VEL
LIN {X 0,Y 501.494,Z 582.727,A -85,B 0,C 180,E1 6256.126,E2 6256.126} C_VEL
LIN {X 0,Y 504.784,Z 545.793,A -85,B 0,C 180,E1 6258.765,E2 6258.765} C_VEL
LIN {X 0,Y 506.724,Z 517.091,A -85,B 0,C 180,E1 6260.274,E2 6260.274} C_VEL
LIN {X 0,Y 492.236,Z 480.836,A -85,B 0,C 180,E1 6262.819,E2 6262.819} C_VEL
LIN {X 0,Y 490.58,Z 476.03,A -85,B 0,C 180,E1 6263.18,E2 6263.18} C_VEL
LIN {X 0,Y 490.756,Z 476.03,A -85,B 0,C 180,E1 6268.365,E2 6268.365} C_VEL
LIN {X 0,Y 490.716,Z 476.03,A -85,B 0,C 180,E1 6274.406,E2 6274.406} C_VEL
LIN {X 0,Y 490.878,Z 476.03,A -85,B 0,C 180,E1 6279.034,E2 6279.034} C_VEL
LIN {X 0,Y 497.318,Z 503.631,A -85,B 0,C 180,E1 6279.874,E2 6279.874} C_VEL
LIN {X 0,Y 496.472,Z 534.731,A -85,B 0,C 180,E1 6281.148,E2 6281.148} C_VEL
LIN {X 0,Y 495.418,Z 563.83,A -85,B 0,C 180,E1 6283.12,E2 6283.12} C_VEL
LIN {X 0,Y 494.24,Z 589,A -85,B 0,C 180,E1 6285.67,E2 6285.67} C_VEL
LIN {X 0,Y 493.334,Z 608.759,A -85,B 0,C 180,E1 6288.58,E2 6288.58} C_VEL
LIN {X 0,Y 492.673,Z 622.822,A -85,B 0,C 180,E1 6291.604,E2 6291.604} C_VEL
LIN {X 0,Y 492.456,Z 632.123,A -85,B 0,C 180,E1 6294.705,E2 6294.705} C_VEL
LIN {X 0,Y 492.216,Z 637.478,A -85,B 0,C 180,E1 6298.235,E2 6298.235} C_VEL
LIN {X 0,Y 492.283,Z 637.663,A -85,B 0,C 180,E1 6301.76,E2 6301.76} C_VEL
LIN {X 0,Y 492.489,Z 632.662,A -85,B 0,C 180,E1 6305.289,E2 6305.289} C_VEL
LIN {X 0,Y 492.94,Z 621.901,A -85,B 0,C 180,E1 6308.831,E2 6308.831} C_VEL
LIN {X 0,Y 493.737,Z 606.582,A -85,B 0,C 180,E1 6311.942,E2 6311.942} C_VEL
LIN {X 0,Y 494.694,Z 585.749,A -85,B 0,C 180,E1 6314.794,E2 6314.794} C_VEL
LIN {X 0,Y 495.791,Z 561.186,A -85,B 0,C 180,E1 6317.09,E2 6317.09} C_VEL
LIN {X 0,Y 496.608,Z 533.2,A -85,B 0,C 180,E1 6318.832,E2 6318.832} C_VEL
LIN {X 0,Y 497.087,Z 503.296,A -85,B 0,C 180,E1 6319.936,E2 6319.936} C_VEL
LIN {X 0,Y 491.107,Z 476.03,A -85,B 0,C 180,E1 6320.703,E2 6320.703} C_VEL
LIN {X 0,Y 490.712,Z 476.03,A -85,B 0,C 180,E1 6327.565,E2 6327.565} C_VEL
LIN {X 0,Y 490.6,Z 476.03,A -85,B 0,C 180,E1 6333.741,E2 6333.741} C_VEL
LIN {X 0,Y 490.573,Z 476.03,A -85,B 0,C 180,E1 6338.463,E2 6338.463} C_VEL
LIN {X 0,Y 488.014,Z 476.03,A -85,B 0,C 180,E1 6339.969,E2 6339.969} C_VEL
LIN {X 0,Y 482.684,Z 476.03,A -85,B 0,C 180,E1 6342.229,E2 6342.229} C_VEL
LIN {X 0,Y 482.595,Z 476.03,A -85,B 0,C 180,E1 6342.49,E2 6342.49} C_VEL
LIN {X 0,Y 482.62,Z 476.03,A -85,B 0,C 180,E1 6348.837,E2 6348.837} C_VEL
LIN {X 0,Y 482.67,Z 476.608,A -85,B 0,C 180,E1 6351.774,E2 6351.774} C_VEL
LIN {X 0,Y 496.031,Z 505.821,A -85,B 0,C 180,E1 6353.425,E2 6353.425} C_VEL
LIN {X 0,Y 503.232,Z 518.429,A -85,B 0,C 180,E1 6354.226,E2 6354.226} C_VEL
LIN {X 0,Y 501.534,Z 561.609,A -85,B 0,C 180,E1 6355.292,E2 6355.292} C_VEL
LIN {X 0,Y 499.045,Z 601.569,A -85,B 0,C 180,E1 6356.963,E2 6356.963} C_VEL
LIN {X 0,Y 496.157,Z 635.333,A -85,B 0,C 180,E1 6359.004,E2 6359.004} C_VEL
LIN {X 0,Y 492.631,Z 669.803,A -85,B 0,C 180,E1 6361.929,E2 6361.929} C_VEL
LIN {X 0,Y 489.504,Z 699.744,A -85,B 0,C 180,E1 6365.318,E2 6365.318} C_VEL
LIN {X 0,Y 486.765,Z 726.983,A -85,B 0,C 180,E1 6369.397,E2 6369.397} C_VEL
LIN {X 0,Y 485.033,Z 748.296,A -85,B 0,C 180,E1 6373.683,E2 6373.683} C_VEL
LIN {X 0,Y 484.117,Z 763.302,A -85,B 0,C 180,E1 6377.812,E2 6377.812} C_VEL
LIN {X 0,Y 483.803,Z 773.544,A -85,B 0,C 180,E1 6381.904,E2 6381.904} C_VEL
LIN {X 0,Y 483.598,Z 779.935,A -85,B 0,C 180,E1 6386.41,E2 6386.41} C_VEL
LIN {X 0,Y 483.656,Z 781.5,A -85,B 0,C 180,E1 6390,E2 6390} C_VEL
LIN {X 0,Y 483.673,Z 779.935,A -85,B 0,C 180,E1 6393.589,E2 6393.589} C_VEL
LIN {X 0,Y 483.844,Z 773.545,A -85,B 0,C 180,E1 6398.095,E2 6398.095} C_VEL
LIN {X 0,Y 484.254,Z 761.895,A -85,B 0,C 180,E1 6402.642,E2 6402.642} C_VEL
LIN {X 0,Y 485.292,Z 744.313,A -85,B 0,C 180,E1 6407.228,E2 6407.228} C_VEL
LIN {X 0,Y 487.232,Z 721.975,A -85,B 0,C 180,E1 6411.449,E2 6411.449} C_VEL
LIN {X 0,Y 489.98,Z 695.132,A -85,B 0,C 180,E1 6415.268,E2 6415.268} C_VEL
LIN {X 0,Y 493.359,Z 663.584,A -85,B 0,C 180,E1 6418.665,E2 6418.665} C_VEL
LIN {X 0,Y 496.831,Z 629.006,A -85,B 0,C 180,E1 6421.438,E2 6421.438} C_VEL
LIN {X 0,Y 499.754,Z 591.994,A -85,B 0,C 180,E1 6423.523,E2 6423.523} C_VEL
LIN {X 0,Y 502.308,Z 553.104,A -85,B 0,C 180,E1 6424.994,E2 6424.994} C_VEL
LIN {X 0,Y 503.093,Z 518.17,A -85,B 0,C 180,E1 6425.845,E2 6425.845} C_VEL
LIN {X 0,Y 489.668,Z 494.634,A -85,B 0,C 180,E1 6427.417,E2 6427.417} C_VEL
LIN {X 0,Y 482.965,Z 477.901,A -85,B 0,C 180,E1 6428.404,E2 6428.404} C_VEL
LIN {X 0,Y 482.729,Z 476.03,A -85,B 0,C 180,E1 6428.649,E2 6428.649} C_VEL
LIN {X 0,Y 482.665,Z 476.03,A -85,B 0,C 180,E1 6433.829,E2 6433.829} C_VEL
LIN {X 0,Y 482.604,Z 476.03,A -85,B 0,C 180,E1 6438.848,E2 6438.848} C_VEL
LIN {X 0,Y 482.684,Z 476.03,A -85,B 0,C 180,E1 6445.629,E2 6445.629} C_VEL
LIN {X 0,Y 482.707,Z 476.03,A -85,B 0,C 180,E1 6451.938,E2 6451.938} C_VEL
LIN {X 0,Y 482.885,Z 476.03,A -85,B 0,C 180,E1 6457.902,E2 6457.902} C_VEL
LIN {X 0,Y 483.071,Z 476.03,A -85,B 0,C 180,E1 6463.619,E2 6463.619} C_VEL
LIN {X 0,Y 483.179,Z 476.03,A -85,B 0,C 180,E1 6469.166,E2 6469.166} C_VEL
LIN {X 0,Y 483.341,Z 476.03,A -85,B 0,C 180,E1 6474.611,E2 6474.611} C_VEL
LIN {X 0,Y 483.522,Z 476.03,A -85,B 0,C 180,E1 6480.003,E2 6480.003} C_VEL
LIN {X 0,Y 483.385,Z 476.03,A -85,B 0,C 180,E1 6485.394,E2 6485.394} C_VEL
LIN {X 0,Y 483.189,Z 476.03,A -85,B 0,C 180,E1 6490.839,E2 6490.839} C_VEL
LIN {X 0,Y 483.048,Z 476.03,A -85,B 0,C 180,E1 6496.388,E2 6496.388} C_VEL
LIN {X 0,Y 482.971,Z 476.03,A -85,B 0,C 180,E1 6502.1,E2 6502.1} C_VEL
LIN {X 0,Y 482.759,Z 476.03,A -85,B 0,C 180,E1 6508.065,E2 6508.065} C_VEL
LIN {X 0,Y 482.663,Z 476.03,A -85,B 0,C 180,E1 6514.379,E2 6514.379} C_VEL
LIN {X 0,Y 482.691,Z 476.03,A -85,B 0,C 180,E1 6518.856,E2 6518.856} C_VEL
LIN {X 0,Y 482.661,Z 476.03,A -85,B 0,C 180,E1 6523.821,E2 6523.821} C_VEL
LIN {X 0,Y 482.69,Z 476.03,A -85,B 0,C 180,E1 6528.836,E2 6528.836} C_VEL
LIN {X 0,Y 482.608,Z 476.03,A -85,B 0,C 180,E1 6534.657,E2 6534.657} C_VEL
LIN {X 0,Y 482.711,Z 476.03,A -85,B 0,C 180,E1 6539.876,E2 6539.876} C_VEL
LIN {X 0,Y 482.896,Z 476.03,A -85,B 0,C 180,E1 6545.945,E2 6545.945} C_VEL
LIN {X 0,Y 483.061,Z 476.083,A -85,B 0,C 180,E1 6550.144,E2 6550.144} C_VEL
LIN {X 0,Y 497.562,Z 512.15,A -85,B 0,C 180,E1 6552.695,E2 6552.695} C_VEL
LIN {X 0,Y 500,Z 521.84,A -85,B 0,C 180,E1 6553.376,E2 6553.376} C_VEL
LIN {X 0,Y 496.9,Z 558.042,A -85,B 0,C 180,E1 6555.441,E2 6555.441} C_VEL
LIN {X 0,Y 493.202,Z 594.468,A -85,B 0,C 180,E1 6558.378,E2 6558.378} C_VEL
LIN {X 0,Y 489.937,Z 624.945,A -85,B 0,C 180,E1 6561.667,E2 6561.667} C_VEL
LIN {X 0,Y 487.1,Z 653.564,A -85,B 0,C 180,E1 6565.767,E2 6565.767} C_VEL
LIN {X 0,Y 485.134,Z 676.866,A -85,B 0,C 180,E1 6570.305,E2 6570.305} C_VEL
LIN {X 0,Y 484.21,Z 692.399,A -85,B 0,C 180,E1 6574.484,E2 6574.484} C_VEL
LIN {X 0,Y 483.771,Z 703.793,A -85,B 0,C 180,E1 6579.004,E2 6579.004} C_VEL
LIN {X 0,Y 483.502,Z 709.234,A -85,B 0,C 180,E1 6582.663,E2 6582.663} C_VEL
LIN {X 0,Y 483.345,Z 711.395,A -85,B 0,C 180,E1 6586.376,E2 6586.376} C_VEL
LIN {X 0,Y 483.399,Z 710.219,A -85,B 0,C 180,E1 6590.154,E2 6590.154} C_VEL
LIN {X 0,Y 483.748,Z 703.984,A -85,B 0,C 180,E1 6594.814,E2 6594.814} C_VEL
LIN {X 0,Y 484.284,Z 692.448,A -85,B 0,C 180,E1 6599.407,E2 6599.407} C_VEL
LIN {X 0,Y 485.186,Z 676.266,A -85,B 0,C 180,E1 6603.737,E2 6603.737} C_VEL
LIN {X 0,Y 487.084,Z 653.7,A -85,B 0,C 180,E1 6608.119,E2 6608.119} C_VEL
LIN {X 0,Y 489.918,Z 625.344,A -85,B 0,C 180,E1 6612.19,E2 6612.19} C_VEL
LIN {X 0,Y 493.104,Z 595.487,A -85,B 0,C 180,E1 6615.439,E2 6615.439} C_VEL
LIN {X 0,Y 496.676,Z 560.316,A -85,B 0,C 180,E1 6618.311,E2 6618.311} C_VEL
LIN {X 0,Y 499.819,Z 524.168,A -85,B 0,C 180,E1 6620.417,E2 6620.417} C_VEL
LIN {X 0,Y 499.506,Z 518.524,A -85,B 0,C 180,E1 6620.745,E2 6620.745} C_VEL
LIN {X 0,Y 485.04,Z 482.71,A -85,B 0,C 180,E1 6623.342,E2 6623.342} C_VEL
LIN {X 0,Y 482.7,Z 476.03,A -85,B 0,C 180,E1 6623.745,E2 6623.745} C_VEL
LIN {X 0,Y 482.784,Z 476.03,A -85,B 0,C 180,E1 6629.88,E2 6629.88} C_VEL
LIN {X 0,Y 482.803,Z 476.03,A -85,B 0,C 180,E1 6635.939,E2 6635.939} C_VEL
LIN {X 0,Y 482.979,Z 476.03,A -85,B 0,C 180,E1 6638.722,E2 6638.722} C_VEL
LIN {X 0,Y 489.75,Z 505.894,A -85,B 0,C 180,E1 6639.649,E2 6639.649} C_VEL
LIN {X 0,Y 488.931,Z 537.227,A -85,B 0,C 180,E1 6640.985,E2 6640.985} C_VEL
LIN {X 0,Y 487.821,Z 565.655,A -85,B 0,C 180,E1 6642.965,E2 6642.965} C_VEL
LIN {X 0,Y 486.587,Z 589.835,A -85,B 0,C 180,E1 6645.45,E2 6645.45} C_VEL
LIN {X 0,Y 485.623,Z 610.48,A -85,B 0,C 180,E1 6648.533,E2 6648.533} C_VEL
LIN {X 0,Y 484.865,Z 625.582,A -85,B 0,C 180,E1 6651.92,E2 6651.92} C_VEL
LIN {X 0,Y 484.571,Z 635.201,A -85,B 0,C 180,E1 6655.517,E2 6655.517} C_VEL
LIN {X 0,Y 484.451,Z 638.77,A -85,B 0,C 180,E1 6658.206,E2 6658.206} C_VEL
LIN {X 0,Y 484.521,Z 639.002,A -85,B 0,C 180,E1 6661.788,E2 6661.788} C_VEL
LIN {X 0,Y 484.759,Z 634.009,A -85,B 0,C 180,E1 6665.374,E2 6665.374} C_VEL
LIN {X 0,Y 485.235,Z 623.195,A -85,B 0,C 180,E1 6668.972,E2 6668.972} C_VEL
LIN {X 0,Y 486.087,Z 607.759,A -85,B 0,C 180,E1 6672.134,E2 6672.134} C_VEL
LIN {X 0,Y 487.106,Z 586.862,A -85,B 0,C 180,E1 6675.017,E2 6675.017} C_VEL
LIN {X 0,Y 488.27,Z 561.89,A -85,B 0,C 180,E1 6677.362,E2 6677.362} C_VEL
LIN {X 0,Y 489.123,Z 533.592,A -85,B 0,C 180,E1 6679.116,E2 6679.116} C_VEL
LIN {X 0,Y 489.59,Z 502.177,A -85,B 0,C 180,E1 6680.249,E2 6680.249} C_VEL
LIN {X 0,Y 483.141,Z 476.03,A -85,B 0,C 180,E1 6680.988,E2 6680.988} C_VEL
LIN {X 0,Y 482.871,Z 476.03,A -85,B 0,C 180,E1 6686.034,E2 6686.034} C_VEL
LIN {X 0,Y 482.677,Z 476.03,A -85,B 0,C 180,E1 6692.221,E2 6692.221} C_VEL
LIN {X 0,Y 482.672,Z 476.03,A -85,B 0,C 180,E1 6698.851,E2 6698.851} C_VEL
LIN {X 0,Y 482.595,Z 476.03,A -85,B 0,C 180,E1 6702.49,E2 6702.49} C_VEL
LIN {X 0,Y 480.059,Z 476.03,A -85,B 0,C 180,E1 6704.024,E2 6704.024} C_VEL
LIN {X 0,Y 474.705,Z 476.03,A -85,B 0,C 180,E1 6706.325,E2 6706.325} C_VEL
LIN {X 0,Y 474.618,Z 476.03,A -85,B 0,C 180,E1 6706.592,E2 6706.592} C_VEL
LIN {X 0,Y 474.728,Z 476.266,A -85,B 0,C 180,E1 6711.037,E2 6711.037} C_VEL
LIN {X 0,Y 490.637,Z 510.685,A -85,B 0,C 180,E1 6713.07,E2 6713.07} C_VEL
LIN {X 0,Y 496.505,Z 520.581,A -85,B 0,C 180,E1 6713.742,E2 6713.742} C_VEL
LIN {X 0,Y 494.536,Z 564.715,A -85,B 0,C 180,E1 6714.933,E2 6714.933} C_VEL
LIN {X 0,Y 491.579,Z 606.228,A -85,B 0,C 180,E1 6716.791,E2 6716.791} C_VEL
LIN {X 0,Y 488.157,Z 644.112,A -85,B 0,C 180,E1 6719.244,E2 6719.244} C_VEL
LIN {X 0,Y 485.071,Z 673.868,A -85,B 0,C 180,E1 6721.889,E2 6721.889} C_VEL
LIN {X 0,Y 481.422,Z 705.186,A -85,B 0,C 180,E1 6725.644,E2 6725.644} C_VEL
LIN {X 0,Y 478.745,Z 731.549,A -85,B 0,C 180,E1 6729.882,E2 6729.882} C_VEL
LIN {X 0,Y 477.059,Z 752.092,A -85,B 0,C 180,E1 6734.349,E2 6734.349} C_VEL
LIN {X 0,Y 476.148,Z 767.222,A -85,B 0,C 180,E1 6739,E2 6739} C_VEL
LIN {X 0,Y 475.838,Z 776.706,A -85,B 0,C 180,E1 6743.605,E2 6743.605} C_VEL
LIN {X 0,Y 475.742,Z 781.108,A -85,B 0,C 180,E1 6748.176,E2 6748.176} C_VEL
LIN {X 0,Y 475.853,Z 781.108,A -85,B 0,C 180,E1 6751.823,E2 6751.823} C_VEL
LIN {X 0,Y 475.83,Z 776.707,A -85,B 0,C 180,E1 6756.394,E2 6756.394} C_VEL
LIN {X 0,Y 476.229,Z 767.224,A -85,B 0,C 180,E1 6760.997,E2 6760.997} C_VEL
LIN {X 0,Y 477.025,Z 752.096,A -85,B 0,C 180,E1 6765.652,E2 6765.652} C_VEL
LIN {X 0,Y 478.796,Z 731.553,A -85,B 0,C 180,E1 6770.115,E2 6770.115} C_VEL
LIN {X 0,Y 481.446,Z 705.342,A -85,B 0,C 180,E1 6774.332,E2 6774.332} C_VEL
LIN {X 0,Y 484.86,Z 675.572,A -85,B 0,C 180,E1 6777.931,E2 6777.931} C_VEL
LIN {X 0,Y 488.182,Z 644.054,A -85,B 0,C 180,E1 6780.768,E2 6780.768} C_VEL
LIN {X 0,Y 491.589,Z 605.88,A -85,B 0,C 180,E1 6783.273,E2 6783.273} C_VEL
LIN {X 0,Y 494.795,Z 564.877,A -85,B 0,C 180,E1 6785.115,E2 6785.115} C_VEL
LIN {X 0,Y 497.048,Z 521.695,A -85,B 0,C 180,E1 6786.274,E2 6786.274} C_VEL
LIN {X 0,Y 484.083,Z 498.859,A -85,B 0,C 180,E1 6787.846,E2 6787.846} C_VEL
LIN {X 0,Y 474.779,Z 476.03,A -85,B 0,C 180,E1 6789.198,E2 6789.198} C_VEL
LIN {X 0,Y 474.648,Z 476.03,A -85,B 0,C 180,E1 6795.437,E2 6795.437} C_VEL
LIN {X 0,Y 474.614,Z 476.03,A -85,B 0,C 180,E1 6800.361,E2 6800.361} C_VEL
LIN {X 0,Y 474.753,Z 476.03,A -85,B 0,C 180,E1 6806.017,E2 6806.017} C_VEL
LIN {X 0,Y 474.807,Z 476.03,A -85,B 0,C 180,E1 6811.429,E2 6811.429} C_VEL
LIN {X 0,Y 474.939,Z 476.03,A -85,B 0,C 180,E1 6817.596,E2 6817.596} C_VEL
LIN {X 0,Y 475.126,Z 476.03,A -85,B 0,C 180,E1 6823.337,E2 6823.337} C_VEL
LIN {X 0,Y 475.251,Z 476.03,A -85,B 0,C 180,E1 6828.983,E2 6828.983} C_VEL
LIN {X 0,Y 475.424,Z 476.03,A -85,B 0,C 180,E1 6834.521,E2 6834.521} C_VEL
LIN {X 0,Y 475.621,Z 476.03,A -85,B 0,C 180,E1 6840.003,E2 6840.003} C_VEL
LIN {X 0,Y 475.471,Z 476.03,A -85,B 0,C 180,E1 6845.484,E2 6845.484} C_VEL
LIN {X 0,Y 475.259,Z 476.03,A -85,B 0,C 180,E1 6851.022,E2 6851.022} C_VEL
LIN {X 0,Y 475.087,Z 476.03,A -85,B 0,C 180,E1 6857.039,E2 6857.039} C_VEL
LIN {X 0,Y 475.037,Z 476.03,A -85,B 0,C 180,E1 6862.489,E2 6862.489} C_VEL
LIN {X 0,Y 474.825,Z 476.03,A -85,B 0,C 180,E1 6868.576,E2 6868.576} C_VEL
LIN {X 0,Y 474.751,Z 476.03,A -85,B 0,C 180,E1 6875.035,E2 6875.035} C_VEL
LIN {X 0,Y 474.689,Z 476.03,A -85,B 0,C 180,E1 6880.047,E2 6880.047} C_VEL
LIN {X 0,Y 474.696,Z 476.03,A -85,B 0,C 180,E1 6885.435,E2 6885.435} C_VEL
LIN {X 0,Y 474.685,Z 476.03,A -85,B 0,C 180,E1 6890.362,E2 6890.362} C_VEL
LIN {X 0,Y 474.673,Z 476.03,A -85,B 0,C 180,E1 6896.031,E2 6896.031} C_VEL
LIN {X 0,Y 474.804,Z 476.03,A -85,B 0,C 180,E1 6901.423,E2 6901.423} C_VEL
LIN {X 0,Y 475.032,Z 476.03,A -85,B 0,C 180,E1 6907.567,E2 6907.567} C_VEL
LIN {X 0,Y 475.07,Z 476.03,A -85,B 0,C 180,E1 6909.418,E2 6909.418} C_VEL
LIN {X 0,Y 490.409,Z 513.666,A -85,B 0,C 180,E1 6912.195,E2 6912.195} C_VEL
LIN {X 0,Y 493.275,Z 523.484,A -85,B 0,C 180,E1 6912.937,E2 6912.937} C_VEL
LIN {X 0,Y 490.051,Z 559.138,A -85,B 0,C 180,E1 6915.004,E2 6915.004} C_VEL
LIN {X 0,Y 486.18,Z 593.901,A -85,B 0,C 180,E1 6917.865,E2 6917.865} C_VEL
LIN {X 0,Y 482.586,Z 624.96,A -85,B 0,C 180,E1 6921.257,E2 6921.257} C_VEL
LIN {X 0,Y 479.632,Z 652.554,A -85,B 0,C 180,E1 6925.247,E2 6925.247} C_VEL
LIN {X 0,Y 477.509,Z 675.723,A -85,B 0,C 180,E1 6929.773,E2 6929.773} C_VEL
LIN {X 0,Y 476.399,Z 691.886,A -85,B 0,C 180,E1 6934.101,E2 6934.101} C_VEL
LIN {X 0,Y 475.952,Z 702.506,A -85,B 0,C 180,E1 6938.231,E2 6938.231} C_VEL
LIN {X 0,Y 475.57,Z 709.544,A -85,B 0,C 180,E1 6942.878,E2 6942.878} C_VEL
LIN {X 0,Y 475.392,Z 711.471,A -85,B 0,C 180,E1 6947.162,E2 6947.162} C_VEL
LIN {X 0,Y 475.565,Z 709.055,A -85,B 0,C 180,E1 6951.478,E2 6951.478} C_VEL
LIN {X 0,Y 475.926,Z 702.165,A -85,B 0,C 180,E1 6955.848,E2 6955.848} C_VEL
LIN {X 0,Y 476.597,Z 689.455,A -85,B 0,C 180,E1 6960.552,E2 6960.552} C_VEL
LIN {X 0,Y 477.89,Z 670.932,A -85,B 0,C 180,E1 6965.207,E2 6965.207} C_VEL
LIN {X 0,Y 480.275,Z 646.524,A -85,B 0,C 180,E1 6969.624,E2 6969.624} C_VEL
LIN {X 0,Y 483.247,Z 619.236,A -85,B 0,C 180,E1 6973.354,E2 6973.354} C_VEL
LIN {X 0,Y 487.258,Z 585.01,A -85,B 0,C 180,E1 6976.872,E2 6976.872} C_VEL
LIN {X 0,Y 490.97,Z 549.015,A -85,B 0,C 180,E1 6979.567,E2 6979.567} C_VEL
LIN {X 0,Y 493.07,Z 522.331,A -85,B 0,C 180,E1 6981.04,E2 6981.04} C_VEL
LIN {X 0,Y 479.33,Z 487.454,A -85,B 0,C 180,E1 6983.667,E2 6983.667} C_VEL
LIN {X 0,Y 474.774,Z 476.03,A -85,B 0,C 180,E1 6984.471,E2 6984.471} C_VEL
LIN {X 0,Y 474.858,Z 476.03,A -85,B 0,C 180,E1 6989.42,E2 6989.42} C_VEL
LIN {X 0,Y 474.914,Z 476.03,A -85,B 0,C 180,E1 6995.513,E2 6995.513} C_VEL
LIN {X 0,Y 475.023,Z 476.047,A -85,B 0,C 180,E1 6998.414,E2 6998.414} C_VEL
LIN {X 0,Y 482.242,Z 506.81,A -85,B 0,C 180,E1 6999.375,E2 6999.375} C_VEL
LIN {X 0,Y 481.415,Z 537.75,A -85,B 0,C 180,E1 7000.706,E2 7000.706} C_VEL
LIN {X 0,Y 480.253,Z 566.106,A -85,B 0,C 180,E1 7002.688,E2 7002.688} C_VEL
LIN {X 0,Y 478.968,Z 589.994,A -85,B 0,C 180,E1 7005.143,E2 7005.143} C_VEL
LIN {X 0,Y 477.986,Z 610.122,A -85,B 0,C 180,E1 7008.116,E2 7008.116} C_VEL
LIN {X 0,Y 477.198,Z 625.012,A -85,B 0,C 180,E1 7011.33,E2 7011.33} C_VEL
LIN {X 0,Y 476.925,Z 634.54,A -85,B 0,C 180,E1 7014.532,E2 7014.532} C_VEL
LIN {X 0,Y 476.693,Z 640.064,A -85,B 0,C 180,E1 7018.177,E2 7018.177} C_VEL
LIN {X 0,Y 476.762,Z 640.347,A -85,B 0,C 180,E1 7021.817,E2 7021.817} C_VEL
LIN {X 0,Y 477.003,Z 635.363,A -85,B 0,C 180,E1 7025.461,E2 7025.461} C_VEL
LIN {X 0,Y 477.558,Z 624.488,A -85,B 0,C 180,E1 7029.118,E2 7029.118} C_VEL
LIN {X 0,Y 478.471,Z 608.972,A -85,B 0,C 180,E1 7032.33,E2 7032.33} C_VEL
LIN {X 0,Y 479.537,Z 587.978,A -85,B 0,C 180,E1 7035.251,E2 7035.251} C_VEL
LIN {X 0,Y 480.784,Z 562.624,A -85,B 0,C 180,E1 7037.641,E2 7037.641} C_VEL
LIN {X 0,Y 481.642,Z 533.898,A -85,B 0,C 180,E1 7039.421,E2 7039.421} C_VEL
LIN {X 0,Y 481.943,Z 502.65,A -85,B 0,C 180,E1 7040.541,E2 7040.541} C_VEL
LIN {X 0,Y 475.23,Z 476.03,A -85,B 0,C 180,E1 7041.342,E2 7041.342} C_VEL
LIN {X 0,Y 474.858,Z 476.03,A -85,B 0,C 180,E1 7046.772,E2 7046.772} C_VEL
LIN {X 0,Y 474.692,Z 476.03,A -85,B 0,C 180,E1 7052.831,E2 7052.831} C_VEL
LIN {X 0,Y 474.729,Z 476.03,A -85,B 0,C 180,E1 7057.294,E2 7057.294} C_VEL
LIN {X 0,Y 474.706,Z 476.03,A -85,B 0,C 180,E1 7062.81,E2 7062.81} C_VEL
LIN {X 0,Y 474.618,Z 476.03,A -85,B 0,C 180,E1 7066.592,E2 7066.592} C_VEL
LIN {X 0,Y 470.653,Z 476.03,A -85,B 0,C 180,E1 7067.936,E2 7067.936} C_VEL
LIN {X 0,Y 466.678,Z 476.03,A -85,B 0,C 180,E1 7069.304,E2 7069.304} C_VEL
LIN {X 0,Y 466.723,Z 476.03,A -85,B 0,C 180,E1 7070.246,E2 7070.246} C_VEL
LIN {X 0,Y 471.144,Z 485.815,A -85,B 0,C 180,E1 7070.869,E2 7070.869} C_VEL
LIN {X 0,Y 485.857,Z 516.538,A -85,B 0,C 180,E1 7072.79,E2 7072.79} C_VEL
LIN {X 0,Y 490.045,Z 523.444,A -85,B 0,C 180,E1 7073.287,E2 7073.287} C_VEL
LIN {X 0,Y 487.602,Z 566.62,A -85,B 0,C 180,E1 7074.529,E2 7074.529} C_VEL
LIN {X 0,Y 484.301,Z 608.53,A -85,B 0,C 180,E1 7076.495,E2 7076.495} C_VEL
LIN {X 0,Y 480.638,Z 646.431,A -85,B 0,C 180,E1 7079.048,E2 7079.048} C_VEL
LIN {X 0,Y 477.092,Z 680.291,A -85,B 0,C 180,E1 7082.152,E2 7082.152} C_VEL
LIN {X 0,Y 473.612,Z 708.736,A -85,B 0,C 180,E1 7085.745,E2 7085.745} C_VEL
LIN {X 0,Y 470.89,Z 734.04,A -85,B 0,C 180,E1 7090.023,E2 7090.023} C_VEL
LIN {X 0,Y 469.166,Z 753.881,A -85,B 0,C 180,E1 7094.559,E2 7094.559} C_VEL
LIN {X 0,Y 468.238,Z 768.909,A -85,B 0,C 180,E1 7099.492,E2 7099.492} C_VEL
LIN {X 0,Y 467.879,Z 777.972,A -85,B 0,C 180,E1 7104.428,E2 7104.428} C_VEL
LIN {X 0,Y 467.857,Z 781.107,A -85,B 0,C 180,E1 7108.145,E2 7108.145} C_VEL
LIN {X 0,Y 467.952,Z 781.107,A -85,B 0,C 180,E1 7111.854,E2 7111.854} C_VEL
LIN {X 0,Y 467.932,Z 776.706,A -85,B 0,C 180,E1 7116.502,E2 7116.502} C_VEL
LIN {X 0,Y 468.354,Z 767.223,A -85,B 0,C 180,E1 7121.184,E2 7121.184} C_VEL
LIN {X 0,Y 469.235,Z 752.095,A -85,B 0,C 180,E1 7125.919,E2 7125.919} C_VEL
LIN {X 0,Y 471.122,Z 731.552,A -85,B 0,C 180,E1 7130.457,E2 7130.457} C_VEL
LIN {X 0,Y 473.887,Z 706.713,A -85,B 0,C 180,E1 7134.542,E2 7134.542} C_VEL
LIN {X 0,Y 477.225,Z 678.589,A -85,B 0,C 180,E1 7138.032,E2 7138.032} C_VEL
LIN {X 0,Y 480.998,Z 643.908,A -85,B 0,C 180,E1 7141.184,E2 7141.184} C_VEL
LIN {X 0,Y 484.68,Z 605.691,A -85,B 0,C 180,E1 7143.743,E2 7143.743} C_VEL
LIN {X 0,Y 488.192,Z 564.543,A -85,B 0,C 180,E1 7145.626,E2 7145.626} C_VEL
LIN {X 0,Y 490.049,Z 523.982,A -85,B 0,C 180,E1 7146.808,E2 7146.808} C_VEL
LIN {X 0,Y 478.869,Z 503.804,A -85,B 0,C 180,E1 7148.241,E2 7148.241} C_VEL
LIN {X 0,Y 468.97,Z 481.436,A -85,B 0,C 180,E1 7149.625,E2 7149.625} C_VEL
LIN {X 0,Y 466.819,Z 476.03,A -85,B 0,C 180,E1 7150.001,E2 7150.001} C_VEL
LIN {X 0,Y 466.734,Z 476.03,A -85,B 0,C 180,E1 7155.536,E2 7155.536} C_VEL
LIN {X 0,Y 466.687,Z 476.03,A -85,B 0,C 180,E1 7161.951,E2 7161.951} C_VEL
LIN {X 0,Y 466.848,Z 476.03,A -85,B 0,C 180,E1 7168.746,E2 7168.746} C_VEL
LIN {X 0,Y 466.967,Z 476.03,A -85,B 0,C 180,E1 7175.214,E2 7175.214} C_VEL
LIN {X 0,Y 467.113,Z 476.03,A -85,B 0,C 180,E1 7181.091,E2 7181.091} C_VEL
LIN {X 0,Y 467.28,Z 476.03,A -85,B 0,C 180,E1 7186.894,E2 7186.894} C_VEL
LIN {X 0,Y 467.413,Z 476.03,A -85,B 0,C 180,E1 7192.558,E2 7192.558} C_VEL
LIN {X 0,Y 467.636,Z 476.03,A -85,B 0,C 180,E1 7198.148,E2 7198.148} C_VEL
LIN {X 0,Y 467.548,Z 476.03,A -85,B 0,C 180,E1 7203.716,E2 7203.716} C_VEL
LIN {X 0,Y 467.366,Z 476.03,A -85,B 0,C 180,E1 7209.324,E2 7209.324} C_VEL
LIN {X 0,Y 467.213,Z 476.03,A -85,B 0,C 180,E1 7215.028,E2 7215.028} C_VEL
LIN {X 0,Y 467.115,Z 476.03,A -85,B 0,C 180,E1 7220.89,E2 7220.89} C_VEL
LIN {X 0,Y 466.965,Z 476.03,A -85,B 0,C 180,E1 7226.998,E2 7226.998} C_VEL
LIN {X 0,Y 466.81,Z 476.03,A -85,B 0,C 180,E1 7233.464,E2 7233.464} C_VEL
LIN {X 0,Y 466.748,Z 476.03,A -85,B 0,C 180,E1 7240.451,E2 7240.451} C_VEL
LIN {X 0,Y 466.812,Z 476.03,A -85,B 0,C 180,E1 7247.068,E2 7247.068} C_VEL
LIN {X 0,Y 466.727,Z 476.03,A -85,B 0,C 180,E1 7251.948,E2 7251.948} C_VEL
LIN {X 0,Y 466.768,Z 476.03,A -85,B 0,C 180,E1 7258.734,E2 7258.734} C_VEL
LIN {X 0,Y 467.062,Z 476.03,A -85,B 0,C 180,E1 7265.187,E2 7265.187} C_VEL
LIN {X 0,Y 467.179,Z 476.702,A -85,B 0,C 180,E1 7268.752,E2 7268.752} C_VEL
LIN {X 0,Y 482.132,Z 512.022,A -85,B 0,C 180,E1 7271.424,E2 7271.424} C_VEL
LIN {X 0,Y 486.509,Z 526.052,A -85,B 0,C 180,E1 7272.533,E2 7272.533} C_VEL
LIN {X 0,Y 483.047,Z 561.721,A -85,B 0,C 180,E1 7274.665,E2 7274.665} C_VEL
LIN {X 0,Y 479.004,Z 596.096,A -85,B 0,C 180,E1 7277.565,E2 7277.565} C_VEL
LIN {X 0,Y 475.07,Z 626.684,A -85,B 0,C 180,E1 7281.059,E2 7281.059} C_VEL
LIN {X 0,Y 471.893,Z 654.21,A -85,B 0,C 180,E1 7285.169,E2 7285.169} C_VEL
LIN {X 0,Y 469.678,Z 676.771,A -85,B 0,C 180,E1 7289.721,E2 7289.721} C_VEL
LIN {X 0,Y 468.527,Z 692.712,A -85,B 0,C 180,E1 7294.17,E2 7294.17} C_VEL
LIN {X 0,Y 468.042,Z 703.071,A -85,B 0,C 180,E1 7298.371,E2 7298.371} C_VEL
LIN {X 0,Y 467.629,Z 709.814,A -85,B 0,C 180,E1 7303.1,E2 7303.1} C_VEL
LIN {X 0,Y 467.504,Z 711.5,A -85,B 0,C 180,E1 7306.947,E2 7306.947} C_VEL
LIN {X 0,Y 467.703,Z 708.72,A -85,B 0,C 180,E1 7311.858,E2 7311.858} C_VEL
LIN {X 0,Y 468.096,Z 701.29,A -85,B 0,C 180,E1 7316.432,E2 7316.432} C_VEL
LIN {X 0,Y 468.833,Z 688.338,A -85,B 0,C 180,E1 7321.113,E2 7321.113} C_VEL
LIN {X 0,Y 470.285,Z 670.15,A -85,B 0,C 180,E1 7325.687,E2 7325.687} C_VEL
LIN {X 0,Y 472.987,Z 644.818,A -85,B 0,C 180,E1 7330.28,E2 7330.28} C_VEL
LIN {X 0,Y 476.367,Z 616.332,A -85,B 0,C 180,E1 7334.143,E2 7334.143} C_VEL
LIN {X 0,Y 480.405,Z 584.635,A -85,B 0,C 180,E1 7337.418,E2 7337.418} C_VEL
LIN {X 0,Y 484.225,Z 549.627,A -85,B 0,C 180,E1 7340.051,E2 7340.051} C_VEL
LIN {X 0,Y 486.163,Z 524.509,A -85,B 0,C 180,E1 7341.473,E2 7341.473} C_VEL
LIN {X 0,Y 472.367,Z 489.358,A -85,B 0,C 180,E1 7344.197,E2 7344.197} C_VEL
LIN {X 0,Y 466.853,Z 476.03,A -85,B 0,C 180,E1 7345.092,E2 7345.092} C_VEL
LIN {X 0,Y 466.9,Z 476.03,A -85,B 0,C 180,E1 7351.115,E2 7351.115} C_VEL
LIN {X 0,Y 467.103,Z 476.03,A -85,B 0,C 180,E1 7358.077,E2 7358.077} C_VEL
LIN {X 0,Y 474.731,Z 507.82,A -85,B 0,C 180,E1 7359.099,E2 7359.099} C_VEL
LIN {X 0,Y 473.905,Z 538.786,A -85,B 0,C 180,E1 7360.449,E2 7360.449} C_VEL
LIN {X 0,Y 472.669,Z 567.911,A -85,B 0,C 180,E1 7362.522,E2 7362.522} C_VEL
LIN {X 0,Y 471.309,Z 592.384,A -85,B 0,C 180,E1 7365.106,E2 7365.106} C_VEL
LIN {X 0,Y 470.249,Z 612.361,A -85,B 0,C 180,E1 7368.153,E2 7368.153} C_VEL
LIN {X 0,Y 469.39,Z 627.802,A -85,B 0,C 180,E1 7371.651,E2 7371.651} C_VEL
LIN {X 0,Y 469.056,Z 637.66,A -85,B 0,C 180,E1 7375.369,E2 7375.369} C_VEL
LIN {X 0,Y 468.917,Z 641.358,A -85,B 0,C 180,E1 7378.147,E2 7378.147} C_VEL
LIN {X 0,Y 468.989,Z 641.695,A -85,B 0,C 180,E1 7381.847,E2 7381.847} C_VEL
LIN {X 0,Y 469.275,Z 636.724,A -85,B 0,C 180,E1 7385.551,E2 7385.551} C_VEL
LIN {X 0,Y 469.882,Z 625.821,A -85,B 0,C 180,E1 7389.268,E2 7389.268} C_VEL
LIN {X 0,Y 470.847,Z 610.201,A -85,B 0,C 180,E1 7392.533,E2 7392.533} C_VEL
LIN {X 0,Y 471.942,Z 589.996,A -85,B 0,C 180,E1 7395.393,E2 7395.393} C_VEL
LIN {X 0,Y 473.246,Z 564.934,A -85,B 0,C 180,E1 7397.811,E2 7397.811} C_VEL
LIN {X 0,Y 474.136,Z 536.606,A -85,B 0,C 180,E1 7399.616,E2 7399.616} C_VEL
LIN {X 0,Y 474.572,Z 507.365,A -85,B 0,C 180,E1 7400.724,E2 7400.724} C_VEL
LIN {X 0,Y 467.266,Z 476.03,A -85,B 0,C 180,E1 7401.738,E2 7401.738} C_VEL
LIN {X 0,Y 466.943,Z 476.03,A -85,B 0,C 180,E1 7406.993,E2 7406.993} C_VEL
LIN {X 0,Y 466.762,Z 476.03,A -85,B 0,C 180,E1 7413.461,E2 7413.461} C_VEL
LIN {X 0,Y 466.76,Z 476.03,A -85,B 0,C 180,E1 7420.442,E2 7420.442} C_VEL
LIN {X 0,Y 466.772,Z 476.03,A -85,B 0,C 180,E1 7427.062,E2 7427.062} C_VEL
LIN {X 0,Y 466.678,Z 476.03,A -85,B 0,C 180,E1 7429.304,E2 7429.304} C_VEL
LIN {X 0,Y 467.347,Z 479.025,A -85,B 0,C 180,E1 7430.069,E2 7430.069} C_VEL
LIN {X 0,Y 469.43,Z 489.572,A -85,B 0,C 180,E1 7430.771,E2 7430.771} C_VEL
LIN {X 0,Y 472.813,Z 506.091,A -85,B 0,C 180,E1 7431.424,E2 7431.424} C_VEL
LIN {X 0,Y 481.719,Z 523.54,A -85,B 0,C 180,E1 7432.616,E2 7432.616} C_VEL
LIN {X 0,Y 483.4,Z 527.919,A -85,B 0,C 180,E1 7432.87,E2 7432.87} C_VEL
LIN {X 0,Y 480.529,Z 570.026,A -85,B 0,C 180,E1 7434.182,E2 7434.182} C_VEL
LIN {X 0,Y 477.041,Z 610.386,A -85,B 0,C 180,E1 7436.173,E2 7436.173} C_VEL
LIN {X 0,Y 473.165,Z 647.8,A -85,B 0,C 180,E1 7438.781,E2 7438.781} C_VEL
LIN {X 0,Y 469.49,Z 681.141,A -85,B 0,C 180,E1 7441.924,E2 7441.924} C_VEL
LIN {X 0,Y 465.968,Z 710.477,A -85,B 0,C 180,E1 7445.6,E2 7445.6} C_VEL
LIN {X 0,Y 463.121,Z 735.24,A -85,B 0,C 180,E1 7449.923,E2 7449.923} C_VEL
LIN {X 0,Y 461.353,Z 753.882,A -85,B 0,C 180,E1 7454.29,E2 7454.29} C_VEL
LIN {X 0,Y 460.391,Z 768.411,A -85,B 0,C 180,E1 7459.099,E2 7459.099} C_VEL
LIN {X 0,Y 460.04,Z 776.704,A -85,B 0,C 180,E1 7463.385,E2 7463.385} C_VEL
LIN {X 0,Y 459.952,Z 781.106,A -85,B 0,C 180,E1 7468.113,E2 7468.113} C_VEL
LIN {X 0,Y 460.046,Z 781.106,A -85,B 0,C 180,E1 7471.886,E2 7471.886} C_VEL
LIN {X 0,Y 460.039,Z 776.705,A -85,B 0,C 180,E1 7476.615,E2 7476.615} C_VEL
LIN {X 0,Y 460.506,Z 767.222,A -85,B 0,C 180,E1 7481.377,E2 7481.377} C_VEL
LIN {X 0,Y 461.473,Z 752.093,A -85,B 0,C 180,E1 7486.194,E2 7486.194} C_VEL
LIN {X 0,Y 463.505,Z 731.55,A -85,B 0,C 180,E1 7490.808,E2 7490.808} C_VEL
LIN {X 0,Y 466.479,Z 706.614,A -85,B 0,C 180,E1 7494.958,E2 7494.958} C_VEL
LIN {X 0,Y 470.187,Z 675.424,A -85,B 0,C 180,E1 7498.713,E2 7498.713} C_VEL
LIN {X 0,Y 474.249,Z 639.886,A -85,B 0,C 180,E1 7501.911,E2 7501.911} C_VEL
LIN {X 0,Y 478.134,Z 601.795,A -85,B 0,C 180,E1 7504.427,E2 7504.427} C_VEL
LIN {X 0,Y 481.926,Z 560.803,A -85,B 0,C 180,E1 7506.267,E2 7506.267} C_VEL
LIN {X 0,Y 483.579,Z 527.498,A -85,B 0,C 180,E1 7507.277,E2 7507.277} C_VEL
LIN {X 0,Y 472.689,Z 506.594,A -85,B 0,C 180,E1 7508.769,E2 7508.769} C_VEL
LIN {X 0,Y 463.604,Z 486.229,A -85,B 0,C 180,E1 7510.072,E2 7510.072} C_VEL
LIN {X 0,Y 458.917,Z 476.906,A -85,B 0,C 180,E1 7510.738,E2 7510.738} C_VEL
LIN {X 0,Y 458.857,Z 476.03,A -85,B 0,C 180,E1 7510.934,E2 7510.934} C_VEL
LIN {X 0,Y 458.812,Z 476.03,A -85,B 0,C 180,E1 7516.553,E2 7516.553} C_VEL
LIN {X 0,Y 458.768,Z 476.03,A -85,B 0,C 180,E1 7522.381,E2 7522.381} C_VEL
LIN {X 0,Y 458.939,Z 476.03,A -85,B 0,C 180,E1 7529.068,E2 7529.068} C_VEL
LIN {X 0,Y 458.987,Z 476.03,A -85,B 0,C 180,E1 7534.611,E2 7534.611} C_VEL
LIN {X 0,Y 459.207,Z 476.03,A -85,B 0,C 180,E1 7540.752,E2 7540.752} C_VEL
LIN {X 0,Y 459.358,Z 476.03,A -85,B 0,C 180,E1 7546.664,E2 7546.664} C_VEL
LIN {X 0,Y 459.497,Z 476.03,A -85,B 0,C 180,E1 7552.429,E2 7552.429} C_VEL
LIN {X 0,Y 459.734,Z 476.03,A -85,B 0,C 180,E1 7558.116,E2 7558.116} C_VEL
LIN {X 0,Y 459.64,Z 476.03,A -85,B 0,C 180,E1 7563.78,E2 7563.78} C_VEL
LIN {X 0,Y 459.443,Z 476.03,A -85,B 0,C 180,E1 7569.487,E2 7569.487} C_VEL
LIN {X 0,Y 459.278,Z 476.03,A -85,B 0,C 180,E1 7575.294,E2 7575.294} C_VEL
LIN {X 0,Y 459.166,Z 476.03,A -85,B 0,C 180,E1 7581.269,E2 7581.269} C_VEL
LIN {X 0,Y 459.01,Z 476.03,A -85,B 0,C 180,E1 7587.505,E2 7587.505} C_VEL
LIN {X 0,Y 458.829,Z 476.03,A -85,B 0,C 180,E1 7594.413,E2 7594.413} C_VEL
LIN {X 0,Y 458.867,Z 476.03,A -85,B 0,C 180,E1 7600.631,E2 7600.631} C_VEL
LIN {X 0,Y 458.875,Z 476.03,A -85,B 0,C 180,E1 7606.545,E2 7606.545} C_VEL
LIN {X 0,Y 458.793,Z 476.03,A -85,B 0,C 180,E1 7612.377,E2 7612.377} C_VEL
LIN {X 0,Y 458.854,Z 476.03,A -85,B 0,C 180,E1 7619.085,E2 7619.085} C_VEL
LIN {X 0,Y 459.068,Z 476.03,A -85,B 0,C 180,E1 7624.611,E2 7624.611} C_VEL
LIN {X 0,Y 459.234,Z 476.03,A -85,B 0,C 180,E1 7627.973,E2 7627.973} C_VEL
LIN {X 0,Y 475.342,Z 514.273,A -85,B 0,C 180,E1 7630.957,E2 7630.957} C_VEL
LIN {X 0,Y 479.666,Z 529.488,A -85,B 0,C 180,E1 7632.159,E2 7632.159} C_VEL
LIN {X 0,Y 476.053,Z 564.308,A -85,B 0,C 180,E1 7634.315,E2 7634.315} C_VEL
LIN {X 0,Y 471.823,Z 598.237,A -85,B 0,C 180,E1 7637.255,E2 7637.255} C_VEL
LIN {X 0,Y 467.808,Z 627.542,A -85,B 0,C 180,E1 7640.687,E2 7640.687} C_VEL
LIN {X 0,Y 464.146,Z 655.797,A -85,B 0,C 180,E1 7645.088,E2 7645.088} C_VEL
LIN {X 0,Y 461.837,Z 678.013,A -85,B 0,C 180,E1 7649.716,E2 7649.716} C_VEL
LIN {X 0,Y 460.644,Z 693.54,A -85,B 0,C 180,E1 7654.242,E2 7654.242} C_VEL
LIN {X 0,Y 460.083,Z 704.838,A -85,B 0,C 180,E1 7659.153,E2 7659.153} C_VEL
LIN {X 0,Y 459.714,Z 710.045,A -85,B 0,C 180,E1 7663.33,E2 7663.33} C_VEL
LIN {X 0,Y 459.584,Z 711.457,A -85,B 0,C 180,E1 7667.248,E2 7667.248} C_VEL
LIN {X 0,Y 459.744,Z 709.47,A -85,B 0,C 180,E1 7671.24,E2 7671.24} C_VEL
LIN {X 0,Y 460.091,Z 703.765,A -85,B 0,C 180,E1 7675.33,E2 7675.33} C_VEL
LIN {X 0,Y 460.702,Z 693.226,A -85,B 0,C 180,E1 7679.777,E2 7679.777} C_VEL
LIN {X 0,Y 461.9,Z 676.956,A -85,B 0,C 180,E1 7684.445,E2 7684.445} C_VEL
LIN {X 0,Y 464.361,Z 654.05,A -85,B 0,C 180,E1 7689.142,E2 7689.142} C_VEL
LIN {X 0,Y 468.248,Z 624.438,A -85,B 0,C 180,E1 7693.644,E2 7693.644} C_VEL
LIN {X 0,Y 472.333,Z 594.038,A -85,B 0,C 180,E1 7697.071,E2 7697.071} C_VEL
LIN {X 0,Y 476.425,Z 560.68,A -85,B 0,C 180,E1 7699.849,E2 7699.849} C_VEL
LIN {X 0,Y 479.548,Z 527.631,A -85,B 0,C 180,E1 7701.838,E2 7701.838} C_VEL
LIN {X 0,Y 465.96,Z 492.545,A -85,B 0,C 180,E1 7704.65,E2 7704.65} C_VEL
LIN {X 0,Y 458.922,Z 476.03,A -85,B 0,C 180,E1 7705.883,E2 7705.883} C_VEL
LIN {X 0,Y 458.964,Z 476.03,A -85,B 0,C 180,E1 7712.492,E2 7712.492} C_VEL
LIN {X 0,Y 459.187,Z 476.03,A -85,B 0,C 180,E1 7717.718,E2 7717.718} C_VEL
LIN {X 0,Y 467.251,Z 508.539,A -85,B 0,C 180,E1 7718.812,E2 7718.812} C_VEL
LIN {X 0,Y 466.353,Z 540.563,A -85,B 0,C 180,E1 7720.234,E2 7720.234} C_VEL
LIN {X 0,Y 465.042,Z 569.617,A -85,B 0,C 180,E1 7722.348,E2 7722.348} C_VEL
LIN {X 0,Y 463.662,Z 593.045,A -85,B 0,C 180,E1 7724.854,E2 7724.854} C_VEL
LIN {X 0,Y 462.558,Z 613.263,A -85,B 0,C 180,E1 7727.953,E2 7727.953} C_VEL
LIN {X 0,Y 461.637,Z 628.898,A -85,B 0,C 180,E1 7731.51,E2 7731.51} C_VEL
LIN {X 0,Y 461.283,Z 638.888,A -85,B 0,C 180,E1 7735.29,E2 7735.29} C_VEL
LIN {X 0,Y 461.158,Z 642.653,A -85,B 0,C 180,E1 7738.116,E2 7738.116} C_VEL
LIN {X 0,Y 461.229,Z 643.055,A -85,B 0,C 180,E1 7741.878,E2 7741.878} C_VEL
LIN {X 0,Y 461.553,Z 638.1,A -85,B 0,C 180,E1 7745.645,E2 7745.645} C_VEL
LIN {X 0,Y 462.201,Z 627.157,A -85,B 0,C 180,E1 7749.424,E2 7749.424} C_VEL
LIN {X 0,Y 463.234,Z 611.477,A -85,B 0,C 180,E1 7752.742,E2 7752.742} C_VEL
LIN {X 0,Y 464.417,Z 591.11,A -85,B 0,C 180,E1 7755.649,E2 7755.649} C_VEL
LIN {X 0,Y 465.799,Z 565.794,A -85,B 0,C 180,E1 7758.105,E2 7758.105} C_VEL
LIN {X 0,Y 466.736,Z 536.879,A -85,B 0,C 180,E1 7759.948,E2 7759.948} C_VEL
LIN {X 0,Y 466.904,Z 505.139,A -85,B 0,C 180,E1 7761.117,E2 7761.117} C_VEL
LIN {X 0,Y 459.316,Z 476.03,A -85,B 0,C 180,E1 7762.047,E2 7762.047} C_VEL
LIN {X 0,Y 458.991,Z 476.03,A -85,B 0,C 180,E1 7767.5,E2 7767.5} C_VEL
LIN {X 0,Y 458.785,Z 476.03,A -85,B 0,C 180,E1 7774.404,E2 7774.404} C_VEL
LIN {X 0,Y 458.881,Z 476.03,A -85,B 0,C 180,E1 7781.286,E2 7781.286} C_VEL
LIN {X 0,Y 458.846,Z 476.03,A -85,B 0,C 180,E1 7786.54,E2 7786.54} C_VEL
LIN {X 0,Y 458.784,Z 476.03,A -85,B 0,C 180,E1 7789.414,E2 7789.414} C_VEL
LIN {X 0,Y 462.835,Z 485.081,A -85,B 0,C 180,E1 7790.022,E2 7790.022} C_VEL
LIN {X 0,Y 472.652,Z 505.624,A -85,B 0,C 180,E1 7791.399,E2 7791.399} C_VEL
LIN {X 0,Y 472.813,Z 506.091,A -85,B 0,C 180,E1 7791.424,E2 7791.424} C_VEL
LIN {X 0,Y 475.57,Z 527.324,A -85,B 0,C 180,E1 7792.199,E2 7792.199} C_VEL
LIN {X 0,Y 476.186,Z 528.447,A -85,B 0,C 180,E1 7792.282,E2 7792.282} C_VEL
LIN {X 0,Y 474.142,Z 565.766,A -85,B 0,C 180,E1 7793.52,E2 7793.52} C_VEL
LIN {X 0,Y 470.595,Z 604.931,A -85,B 0,C 180,E1 7795.402,E2 7795.402} C_VEL
LIN {X 0,Y 466.363,Z 643.233,A -85,B 0,C 180,E1 7798.01,E2 7798.01} C_VEL
LIN {X 0,Y 462.221,Z 679.06,A -85,B 0,C 180,E1 7801.361,E2 7801.361} C_VEL
LIN {X 0,Y 458.451,Z 709.462,A -85,B 0,C 180,E1 7805.173,E2 7805.173} C_VEL
LIN {X 0,Y 455.754,Z 732.818,A -85,B 0,C 180,E1 7809.075,E2 7809.075} C_VEL
LIN {X 0,Y 453.723,Z 752.089,A -85,B 0,C 180,E1 7813.521,E2 7813.521} C_VEL
LIN {X 0,Y 452.553,Z 767.218,A -85,B 0,C 180,E1 7818.419,E2 7818.419} C_VEL
LIN {X 0,Y 452.148,Z 776.703,A -85,B 0,C 180,E1 7823.269,E2 7823.269} C_VEL
LIN {X 0,Y 452.05,Z 781.105,A -85,B 0,C 180,E1 7828.08,E2 7828.08} C_VEL
LIN {X 0,Y 452.166,Z 781.105,A -85,B 0,C 180,E1 7831.919,E2 7831.919} C_VEL
LIN {X 0,Y 452.15,Z 776.704,A -85,B 0,C 180,E1 7836.73,E2 7836.73} C_VEL
LIN {X 0,Y 452.637,Z 767.221,A -85,B 0,C 180,E1 7841.578,E2 7841.578} C_VEL
LIN {X 0,Y 453.729,Z 752.092,A -85,B 0,C 180,E1 7846.478,E2 7846.478} C_VEL
LIN {X 0,Y 455.913,Z 731.549,A -85,B 0,C 180,E1 7851.171,E2 7851.171} C_VEL
LIN {X 0,Y 458.83,Z 706.98,A -85,B 0,C 180,E1 7855.208,E2 7855.208} C_VEL
LIN {X 0,Y 462.838,Z 675.136,A -85,B 0,C 180,E1 7859.124,E2 7859.124} C_VEL
LIN {X 0,Y 467.186,Z 639.347,A -85,B 0,C 180,E1 7862.394,E2 7862.394} C_VEL
LIN {X 0,Y 471.501,Z 600.155,A -85,B 0,C 180,E1 7865.002,E2 7865.002} C_VEL
LIN {X 0,Y 475.432,Z 559.74,A -85,B 0,C 180,E1 7866.835,E2 7866.835} C_VEL
LIN {X 0,Y 477.04,Z 530.794,A -85,B 0,C 180,E1 7867.751,E2 7867.751} C_VEL
LIN {X 0,Y 466.522,Z 509.348,A -85,B 0,C 180,E1 7869.308,E2 7869.308} C_VEL
LIN {X 0,Y 458.498,Z 491.265,A -85,B 0,C 180,E1 7870.495,E2 7870.495} C_VEL
LIN {X 0,Y 451.053,Z 477.375,A -85,B 0,C 180,E1 7871.56,E2 7871.56} C_VEL
LIN {X 0,Y 450.911,Z 476.03,A -85,B 0,C 180,E1 7871.738,E2 7871.738} C_VEL
LIN {X 0,Y 450.817,Z 476.03,A -85,B 0,C 180,E1 7877.808,E2 7877.808} C_VEL
LIN {X 0,Y 450.881,Z 476.03,A -85,B 0,C 180,E1 7883.702,E2 7883.702} C_VEL
LIN {X 0,Y 450.989,Z 476.03,A -85,B 0,C 180,E1 7889.767,E2 7889.767} C_VEL
LIN {X 0,Y 451.086,Z 476.03,A -85,B 0,C 180,E1 7896.252,E2 7896.252} C_VEL
LIN {X 0,Y 451.334,Z 476.03,A -85,B 0,C 180,E1 7902.431,E2 7902.431} C_VEL
LIN {X 0,Y 451.466,Z 476.03,A -85,B 0,C 180,E1 7908.395,E2 7908.395} C_VEL
LIN {X 0,Y 451.671,Z 476.03,A -85,B 0,C 180,E1 7914.232,E2 7914.232} C_VEL
LIN {X 0,Y 451.957,Z 476.03,A -85,B 0,C 180,E1 7920.003,E2 7920.003} C_VEL
LIN {X 0,Y 451.753,Z 476.03,A -85,B 0,C 180,E1 7925.773,E2 7925.773} C_VEL
LIN {X 0,Y 451.468,Z 476.03,A -85,B 0,C 180,E1 7931.611,E2 7931.611} C_VEL
LIN {X 0,Y 451.315,Z 476.03,A -85,B 0,C 180,E1 7937.576,E2 7937.576} C_VEL
LIN {X 0,Y 451.181,Z 476.03,A -85,B 0,C 180,E1 7943.749,E2 7943.749} C_VEL
LIN {X 0,Y 450.963,Z 476.03,A -85,B 0,C 180,E1 7950.241,E2 7950.241} C_VEL
LIN {X 0,Y 450.92,Z 476.03,A -85,B 0,C 180,E1 7957.187,E2 7957.187} C_VEL
LIN {X 0,Y 450.875,Z 476.03,A -85,B 0,C 180,E1 7962.371,E2 7962.371} C_VEL
LIN {X 0,Y 450.897,Z 476.03,A -85,B 0,C 180,E1 7967.81,E2 7967.81} C_VEL
LIN {X 0,Y 450.869,Z 476.03,A -85,B 0,C 180,E1 7973.703,E2 7973.703} C_VEL
LIN {X 0,Y 450.936,Z 476.03,A -85,B 0,C 180,E1 7979.758,E2 7979.758} C_VEL
LIN {X 0,Y 451.17,Z 476.03,A -85,B 0,C 180,E1 7986.252,E2 7986.252} C_VEL
LIN {X 0,Y 451.29,Z 476.167,A -85,B 0,C 180,E1 7987.254,E2 7987.254} C_VEL
LIN {X 0,Y 461.087,Z 498.169,A -85,B 0,C 180,E1 7988.94,E2 7988.94} C_VEL
LIN {X 0,Y 473.067,Z 530.399,A -85,B 0,C 180,E1 7991.648,E2 7991.648} C_VEL
LIN {X 0,Y 469.27,Z 565.351,A -85,B 0,C 180,E1 7993.842,E2 7993.842} C_VEL
LIN {X 0,Y 464.803,Z 599.225,A -85,B 0,C 180,E1 7996.819,E2 7996.819} C_VEL
LIN {X 0,Y 460.307,Z 630.195,A -85,B 0,C 180,E1 8000.534,E2 8000.534} C_VEL
LIN {X 0,Y 456.763,Z 655.108,A -85,B 0,C 180,E1 8004.532,E2 8004.532} C_VEL
LIN {X 0,Y 454.094,Z 678.26,A -85,B 0,C 180,E1 8009.475,E2 8009.475} C_VEL
LIN {X 0,Y 452.751,Z 694.368,A -85,B 0,C 180,E1 8014.316,E2 8014.316} C_VEL
LIN {X 0,Y 452.188,Z 704.992,A -85,B 0,C 180,E1 8019.11,E2 8019.11} C_VEL
LIN {X 0,Y 451.786,Z 710.262,A -85,B 0,C 180,E1 8023.618,E2 8023.618} C_VEL
LIN {X 0,Y 451.649,Z 711.393,A -85,B 0,C 180,E1 8027.561,E2 8027.561} C_VEL
LIN {X 0,Y 451.935,Z 708.343,A -85,B 0,C 180,E1 8032.379,E2 8032.379} C_VEL
LIN {X 0,Y 452.425,Z 699.95,A -85,B 0,C 180,E1 8037.362,E2 8037.362} C_VEL
LIN {X 0,Y 453.411,Z 686.098,A -85,B 0,C 180,E1 8042.297,E2 8042.297} C_VEL
LIN {X 0,Y 455.351,Z 666.722,A -85,B 0,C 180,E1 8047.058,E2 8047.058} C_VEL
LIN {X 0,Y 458.597,Z 642.201,A -85,B 0,C 180,E1 8051.598,E2 8051.598} C_VEL
LIN {X 0,Y 462.877,Z 612.675,A -85,B 0,C 180,E1 8055.625,E2 8055.625} C_VEL
LIN {X 0,Y 467.386,Z 579.481,A -85,B 0,C 180,E1 8058.942,E2 8058.942} C_VEL
LIN {X 0,Y 471.455,Z 544.316,A -85,B 0,C 180,E1 8061.47,E2 8061.47} C_VEL
LIN {X 0,Y 472.485,Z 529.394,A -85,B 0,C 180,E1 8062.329,E2 8062.329} C_VEL
LIN {X 0,Y 458.453,Z 492.963,A -85,B 0,C 180,E1 8065.341,E2 8065.341} C_VEL
LIN {X 0,Y 450.971,Z 476.03,A -85,B 0,C 180,E1 8066.714,E2 8066.714} C_VEL
LIN {X 0,Y 450.994,Z 476.03,A -85,B 0,C 180,E1 8071.963,E2 8071.963} C_VEL
LIN {X 0,Y 451.265,Z 476.03,A -85,B 0,C 180,E1 8077.386,E2 8077.386} C_VEL
LIN {X 0,Y 459.774,Z 509.038,A -85,B 0,C 180,E1 8078.507,E2 8078.507} C_VEL
LIN {X 0,Y 458.857,Z 540.629,A -85,B 0,C 180,E1 8079.912,E2 8079.912} C_VEL
LIN {X 0,Y 457.49,Z 569.946,A -85,B 0,C 180,E1 8082.047,E2 8082.047} C_VEL
LIN {X 0,Y 456.036,Z 593.691,A -85,B 0,C 180,E1 8084.595,E2 8084.595} C_VEL
LIN {X 0,Y 454.851,Z 614.146,A -85,B 0,C 180,E1 8087.746,E2 8087.746} C_VEL
LIN {X 0,Y 453.907,Z 629.971,A -85,B 0,C 180,E1 8091.364,E2 8091.364} C_VEL
LIN {X 0,Y 453.51,Z 640.107,A -85,B 0,C 180,E1 8095.21,E2 8095.21} C_VEL
LIN {X 0,Y 453.377,Z 643.951,A -85,B 0,C 180,E1 8098.083,E2 8098.083} C_VEL
LIN {X 0,Y 453.469,Z 644.416,A -85,B 0,C 180,E1 8101.91,E2 8101.91} C_VEL
LIN {X 0,Y 453.834,Z 639.484,A -85,B 0,C 180,E1 8105.741,E2 8105.741} C_VEL
LIN {X 0,Y 454.533,Z 628.537,A -85,B 0,C 180,E1 8109.584,E2 8109.584} C_VEL
LIN {X 0,Y 455.641,Z 612.767,A -85,B 0,C 180,E1 8112.958,E2 8112.958} C_VEL
LIN {X 0,Y 456.963,Z 591.613,A -85,B 0,C 180,E1 8115.99,E2 8115.99} C_VEL
LIN {X 0,Y 458.353,Z 566.716,A -85,B 0,C 180,E1 8118.41,E2 8118.41} C_VEL
LIN {X 0,Y 459.283,Z 538.686,A -85,B 0,C 180,E1 8120.216,E2 8120.216} C_VEL
LIN {X 0,Y 459.538,Z 506.726,A -85,B 0,C 180,E1 8121.415,E2 8121.415} C_VEL
LIN {X 0,Y 451.335,Z 476.03,A -85,B 0,C 180,E1 8122.451,E2 8122.451} C_VEL
LIN {X 0,Y 450.935,Z 476.03,A -85,B 0,C 180,E1 8129.189,E2 8129.189} C_VEL
LIN {X 0,Y 450.851,Z 476.03,A -85,B 0,C 180,E1 8134.808,E2 8134.808} C_VEL
LIN {X 0,Y 450.911,Z 476.03,A -85,B 0,C 180,E1 8139.636,E2 8139.636} C_VEL
LIN {X 0,Y 450.866,Z 476.03,A -85,B 0,C 180,E1 8145.151,E2 8145.151} C_VEL
LIN {X 0,Y 450.905,Z 476.03,A -85,B 0,C 180,E1 8148.514,E2 8148.514} C_VEL
LIN {X 0,Y 455.2,Z 485.559,A -85,B 0,C 180,E1 8149.216,E2 8149.216} C_VEL
LIN {X 0,Y 465.919,Z 506.867,A -85,B 0,C 180,E1 8150.783,E2 8150.783} C_VEL
LIN {X 0,Y 474.954,Z 526.607,A -85,B 0,C 180,E1 8152.126,E2 8152.126} C_VEL
LIN {X 0,Y 476.186,Z 528.447,A -85,B 0,C 180,E1 8152.282,E2 8152.282} C_VEL
LIN {X 0,Y 477.07,Z 536.006,A -85,B 0,C 180,E1 8152.588,E2 8152.588} C_VEL
LIN {X 0,Y 468.115,Z 559.927,A -85,B 0,C 180,E1 8152.787,E2 8152.787} C_VEL
LIN {X 0,Y 467.763,Z 562.202,A -85,B 0,C 180,E1 8152.865,E2 8152.865} C_VEL
LIN {X 0,Y 463.822,Z 602.785,A -85,B 0,C 180,E1 8154.812,E2 8154.812} C_VEL
LIN {X 0,Y 459.437,Z 640.85,A -85,B 0,C 180,E1 8157.405,E2 8157.405} C_VEL
LIN {X 0,Y 454.929,Z 677.755,A -85,B 0,C 180,E1 8160.872,E2 8160.872} C_VEL
LIN {X 0,Y 450.997,Z 708.078,A -85,B 0,C 180,E1 8164.698,E2 8164.698} C_VEL
LIN {X 0,Y 447.937,Z 733.399,A -85,B 0,C 180,E1 8168.952,E2 8168.952} C_VEL
LIN {X 0,Y 445.967,Z 752.087,A -85,B 0,C 180,E1 8173.226,E2 8173.226} C_VEL
LIN {X 0,Y 444.692,Z 767.217,A -85,B 0,C 180,E1 8178.212,E2 8178.212} C_VEL
LIN {X 0,Y 444.266,Z 776.702,A -85,B 0,C 180,E1 8183.149,E2 8183.149} C_VEL
LIN {X 0,Y 444.144,Z 781.104,A -85,B 0,C 180,E1 8188.046,E2 8188.046} C_VEL
LIN {X 0,Y 444.259,Z 781.104,A -85,B 0,C 180,E1 8191.953,E2 8191.953} C_VEL
LIN {X 0,Y 444.271,Z 776.703,A -85,B 0,C 180,E1 8196.85,E2 8196.85} C_VEL
LIN {X 0,Y 444.802,Z 767.22,A -85,B 0,C 180,E1 8201.785,E2 8201.785} C_VEL
LIN {X 0,Y 445.962,Z 752.091,A -85,B 0,C 180,E1 8206.773,E2 8206.773} C_VEL
LIN {X 0,Y 447.966,Z 733.461,A -85,B 0,C 180,E1 8211.046,E2 8211.046} C_VEL
LIN {X 0,Y 451.049,Z 708.271,A -85,B 0,C 180,E1 8215.315,E2 8215.315} C_VEL
LIN {X 0,Y 455.01,Z 678.63,A -85,B 0,C 180,E1 8219.122,E2 8219.122} C_VEL
LIN {X 0,Y 459.53,Z 643.82,A -85,B 0,C 180,E1 8222.477,E2 8222.477} C_VEL
LIN {X 0,Y 464.147,Z 604.408,A -85,B 0,C 180,E1 8225.255,E2 8225.255} C_VEL
LIN {X 0,Y 468.436,Z 564.211,A -85,B 0,C 180,E1 8227.206,E2 8227.206} C_VEL
LIN {X 0,Y 470.467,Z 533.973,A -85,B 0,C 180,E1 8228.244,E2 8228.244} C_VEL
LIN {X 0,Y 460.364,Z 512.095,A -85,B 0,C 180,E1 8229.841,E2 8229.841} C_VEL
LIN {X 0,Y 452.421,Z 494.507,A -85,B 0,C 180,E1 8231.067,E2 8231.067} C_VEL
LIN {X 0,Y 443.064,Z 477.134,A -85,B 0,C 180,E1 8232.44,E2 8232.44} C_VEL
LIN {X 0,Y 442.958,Z 476.03,A -85,B 0,C 180,E1 8232.486,E2 8232.486} C_VEL
LIN {X 0,Y 442.842,Z 476.03,A -85,B 0,C 180,E1 8239.494,E2 8239.494} C_VEL
LIN {X 0,Y 443.017,Z 476.03,A -85,B 0,C 180,E1 8245.11,E2 8245.11} C_VEL
LIN {X 0,Y 443.047,Z 476.03,A -85,B 0,C 180,E1 8251.421,E2 8251.421} C_VEL
LIN {X 0,Y 443.207,Z 476.03,A -85,B 0,C 180,E1 8257.932,E2 8257.932} C_VEL
LIN {X 0,Y 443.441,Z 476.03,A -85,B 0,C 180,E1 8264.152,E2 8264.152} C_VEL
LIN {X 0,Y 443.668,Z 476.03,A -85,B 0,C 180,E1 8270.179,E2 8270.179} C_VEL
LIN {X 0,Y 443.975,Z 476.03,A -85,B 0,C 180,E1 8276.092,E2 8276.092} C_VEL
LIN {X 0,Y 444.072,Z 476.03,A -85,B 0,C 180,E1 8281.957,E2 8281.957} C_VEL
LIN {X 0,Y 443.695,Z 476.03,A -85,B 0,C 180,E1 8288.26,E2 8288.26} C_VEL
LIN {X 0,Y 443.491,Z 476.03,A -85,B 0,C 180,E1 8293.829,E2 8293.829} C_VEL
LIN {X 0,Y 443.353,Z 476.03,A -85,B 0,C 180,E1 8299.971,E2 8299.971} C_VEL
LIN {X 0,Y 443.17,Z 476.03,A -85,B 0,C 180,E1 8306.37,E2 8306.37} C_VEL
LIN {X 0,Y 442.982,Z 476.03,A -85,B 0,C 180,E1 8313.154,E2 8313.154} C_VEL
LIN {X 0,Y 442.935,Z 476.03,A -85,B 0,C 180,E1 8318.166,E2 8318.166} C_VEL
LIN {X 0,Y 442.914,Z 476.03,A -85,B 0,C 180,E1 8324.12,E2 8324.12} C_VEL
LIN {X 0,Y 442.908,Z 476.03,A -85,B 0,C 180,E1 8329.494,E2 8329.494} C_VEL
LIN {X 0,Y 442.943,Z 476.03,A -85,B 0,C 180,E1 8335.123,E2 8335.123} C_VEL
LIN {X 0,Y 443.051,Z 476.03,A -85,B 0,C 180,E1 8341.416,E2 8341.416} C_VEL
LIN {X 0,Y 443.346,Z 476.759,A -85,B 0,C 180,E1 8346.489,E2 8346.489} C_VEL
LIN {X 0,Y 458.967,Z 511.63,A -85,B 0,C 180,E1 8349.346,E2 8349.346} C_VEL
LIN {X 0,Y 466.208,Z 534.4,A -85,B 0,C 180,E1 8351.29,E2 8351.29} C_VEL
LIN {X 0,Y 461.997,Z 570.937,A -85,B 0,C 180,E1 8353.703,E2 8353.703} C_VEL
LIN {X 0,Y 457.169,Z 604.595,A -85,B 0,C 180,E1 8356.839,E2 8356.839} C_VEL
LIN {X 0,Y 452.61,Z 634.073,A -85,B 0,C 180,E1 8360.56,E2 8360.56} C_VEL
LIN {X 0,Y 448.78,Z 659.665,A -85,B 0,C 180,E1 8364.919,E2 8364.919} C_VEL
LIN {X 0,Y 446.247,Z 679.415,A -85,B 0,C 180,E1 8369.466,E2 8369.466} C_VEL
LIN {X 0,Y 444.856,Z 695.197,A -85,B 0,C 180,E1 8374.392,E2 8374.392} C_VEL
LIN {X 0,Y 444.324,Z 704.734,A -85,B 0,C 180,E1 8378.808,E2 8378.808} C_VEL
LIN {X 0,Y 443.876,Z 710.416,A -85,B 0,C 180,E1 8383.815,E2 8383.815} C_VEL
LIN {X 0,Y 443.746,Z 711.325,A -85,B 0,C 180,E1 8387.884,E2 8387.884} C_VEL
LIN {X 0,Y 444.085,Z 707.79,A -85,B 0,C 180,E1 8392.993,E2 8392.993} C_VEL
LIN {X 0,Y 444.592,Z 699.613,A -85,B 0,C 180,E1 8397.693,E2 8397.693} C_VEL
LIN {X 0,Y 445.791,Z 684.964,A -85,B 0,C 180,E1 8402.918,E2 8402.918} C_VEL
LIN {X 0,Y 448.376,Z 663.15,A -85,B 0,C 180,E1 8408.302,E2 8408.302} C_VEL
LIN {X 0,Y 452.163,Z 637.253,A -85,B 0,C 180,E1 8412.88,E2 8412.88} C_VEL
LIN {X 0,Y 456.613,Z 608.283,A -85,B 0,C 180,E1 8416.659,E2 8416.659} C_VEL
LIN {X 0,Y 460.98,Z 577.437,A -85,B 0,C 180,E1 8419.663,E2 8419.663} C_VEL
LIN {X 0,Y 465.188,Z 541.805,A -85,B 0,C 180,E1 8422.177,E2 8422.177} C_VEL
LIN {X 0,Y 465.782,Z 532.21,A -85,B 0,C 180,E1 8422.739,E2 8422.739} C_VEL
LIN {X 0,Y 452.016,Z 495.683,A -85,B 0,C 180,E1 8425.869,E2 8425.869} C_VEL
LIN {X 0,Y 443.066,Z 476.03,A -85,B 0,C 180,E1 8427.58,E2 8427.58} C_VEL
LIN {X 0,Y 443.107,Z 476.03,A -85,B 0,C 180,E1 8433.626,E2 8433.626} C_VEL
LIN {X 0,Y 443.332,Z 476.571,A -85,B 0,C 180,E1 8437.065,E2 8437.065} C_VEL
LIN {X 0,Y 452.243,Z 510.685,A -85,B 0,C 180,E1 8438.235,E2 8438.235} C_VEL
LIN {X 0,Y 451.339,Z 542.163,A -85,B 0,C 180,E1 8439.671,E2 8439.671} C_VEL
LIN {X 0,Y 449.965,Z 570.224,A -85,B 0,C 180,E1 8441.736,E2 8441.736} C_VEL
LIN {X 0,Y 448.425,Z 594.306,A -85,B 0,C 180,E1 8444.327,E2 8444.327} C_VEL
LIN {X 0,Y 447.16,Z 615.016,A -85,B 0,C 180,E1 8447.532,E2 8447.532} C_VEL
LIN {X 0,Y 446.156,Z 631.041,A -85,B 0,C 180,E1 8451.213,E2 8451.213} C_VEL
LIN {X 0,Y 445.756,Z 641.324,A -85,B 0,C 180,E1 8455.126,E2 8455.126} C_VEL
LIN {X 0,Y 445.618,Z 645.246,A -85,B 0,C 180,E1 8458.05,E2 8458.05} C_VEL
LIN {X 0,Y 445.709,Z 645.789,A -85,B 0,C 180,E1 8461.944,E2 8461.944} C_VEL
LIN {X 0,Y 446.111,Z 640.893,A -85,B 0,C 180,E1 8465.841,E2 8465.841} C_VEL
LIN {X 0,Y 446.696,Z 631.675,A -85,B 0,C 180,E1 8469.262,E2 8469.262} C_VEL
LIN {X 0,Y 447.877,Z 616.813,A -85,B 0,C 180,E1 8472.69,E2 8472.69} C_VEL
LIN {X 0,Y 449.222,Z 596.291,A -85,B 0,C 180,E1 8475.847,E2 8475.847} C_VEL
LIN {X 0,Y 450.711,Z 572.259,A -85,B 0,C 180,E1 8478.353,E2 8478.353} C_VEL
LIN {X 0,Y 451.808,Z 543.652,A -85,B 0,C 180,E1 8480.33,E2 8480.33} C_VEL
LIN {X 0,Y 452.273,Z 512.622,A -85,B 0,C 180,E1 8481.603,E2 8481.603} C_VEL
LIN {X 0,Y 447.63,Z 490.088,A -85,B 0,C 180,E1 8482.322,E2 8482.322} C_VEL
LIN {X 0,Y 443.394,Z 476.03,A -85,B 0,C 180,E1 8482.877,E2 8482.877} C_VEL
LIN {X 0,Y 443.046,Z 476.03,A -85,B 0,C 180,E1 8488.579,E2 8488.579} C_VEL
LIN {X 0,Y 442.929,Z 476.03,A -85,B 0,C 180,E1 8495.523,E2 8495.523} C_VEL
LIN {X 0,Y 442.903,Z 476.03,A -85,B 0,C 180,E1 8501.227,E2 8501.227} C_VEL
LIN {X 0,Y 442.956,Z 476.03,A -85,B 0,C 180,E1 8507.573,E2 8507.573} C_VEL
LIN {X 0,Y 445.451,Z 481.784,A -85,B 0,C 180,E1 8508.019,E2 8508.019} C_VEL
LIN {X 0,Y 459.863,Z 510.016,A -85,B 0,C 180,E1 8510.271,E2 8510.271} C_VEL
LIN {X 0,Y 469.162,Z 531.151,A -85,B 0,C 180,E1 8511.77,E2 8511.77} C_VEL
LIN {X 0,Y 469.865,Z 537.265,A -85,B 0,C 180,E1 8512.034,E2 8512.034} C_VEL
LIN {X 0,Y 467.763,Z 562.202,A -85,B 0,C 180,E1 8512.865,E2 8512.865} C_VEL
LIN {X 0,Y 458.102,Z 592.804,A -85,B 0,C 180,E1 8513.766,E2 8513.766} C_VEL
LIN {X 0,Y 457.803,Z 594.786,A -85,B 0,C 180,E1 8513.864,E2 8513.864} C_VEL
LIN {X 0,Y 452.941,Z 635.583,A -85,B 0,C 180,E1 8516.556,E2 8516.556} C_VEL
LIN {X 0,Y 448.068,Z 672.797,A -85,B 0,C 180,E1 8519.963,E2 8519.963} C_VEL
LIN {X 0,Y 443.806,Z 704.737,A -85,B 0,C 180,E1 8523.931,E2 8523.931} C_VEL
LIN {X 0,Y 440.527,Z 730.579,A -85,B 0,C 180,E1 8528.215,E2 8528.215} C_VEL
LIN {X 0,Y 438.218,Z 751.596,A -85,B 0,C 180,E1 8532.921,E2 8532.921} C_VEL
LIN {X 0,Y 436.928,Z 765.975,A -85,B 0,C 180,E1 8537.491,E2 8537.491} C_VEL
LIN {X 0,Y 436.431,Z 775.221,A -85,B 0,C 180,E1 8542.023,E2 8542.023} C_VEL
LIN {X 0,Y 436.212,Z 779.93,A -85,B 0,C 180,E1 8546.019,E2 8546.019} C_VEL
LIN {X 0,Y 436.273,Z 781.5,A -85,B 0,C 180,E1 8550,E2 8550} C_VEL
LIN {X 0,Y 436.259,Z 779.93,A -85,B 0,C 180,E1 8553.98,E2 8553.98} C_VEL
LIN {X 0,Y 436.566,Z 773.289,A -85,B 0,C 180,E1 8559.119,E2 8559.119} C_VEL
LIN {X 0,Y 437.395,Z 761.153,A -85,B 0,C 180,E1 8564.27,E2 8564.27} C_VEL
LIN {X 0,Y 439.012,Z 743.726,A -85,B 0,C 180,E1 8569.043,E2 8569.043} C_VEL
LIN {X 0,Y 441.946,Z 720.089,A -85,B 0,C 180,E1 8573.738,E2 8573.738} C_VEL
LIN {X 0,Y 445.883,Z 691.068,A -85,B 0,C 180,E1 8578.02,E2 8578.02} C_VEL
LIN {X 0,Y 450.517,Z 657.453,A -85,B 0,C 180,E1 8581.722,E2 8581.722} C_VEL
LIN {X 0,Y 455.551,Z 619.353,A -85,B 0,C 180,E1 8584.806,E2 8584.806} C_VEL
LIN {X 0,Y 460.238,Z 579.099,A -85,B 0,C 180,E1 8587.119,E2 8587.119} C_VEL
LIN {X 0,Y 463.904,Z 537.001,A -85,B 0,C 180,E1 8588.727,E2 8588.727} C_VEL
LIN {X 0,Y 454.381,Z 515.363,A -85,B 0,C 180,E1 8590.346,E2 8590.346} C_VEL
LIN {X 0,Y 446.324,Z 497.484,A -85,B 0,C 180,E1 8591.644,E2 8591.644} C_VEL
LIN {X 0,Y 435.079,Z 477.331,A -85,B 0,C 180,E1 8593.342,E2 8593.342} C_VEL
LIN {X 0,Y 434.969,Z 476.03,A -85,B 0,C 180,E1 8593.471,E2 8593.471} C_VEL
LIN {X 0,Y 434.906,Z 476.03,A -85,B 0,C 180,E1 8599.989,E2 8599.989} C_VEL
LIN {X 0,Y 435.098,Z 476.03,A -85,B 0,C 180,E1 8606.635,E2 8606.635} C_VEL
LIN {X 0,Y 435.162,Z 476.03,A -85,B 0,C 180,E1 8613.113,E2 8613.113} C_VEL
LIN {X 0,Y 435.392,Z 476.03,A -85,B 0,C 180,E1 8619.875,E2 8619.875} C_VEL
LIN {X 0,Y 435.564,Z 476.03,A -85,B 0,C 180,E1 8625.921,E2 8625.921} C_VEL
LIN {X 0,Y 435.793,Z 476.03,A -85,B 0,C 180,E1 8632.015,E2 8632.015} C_VEL
LIN {X 0,Y 436.067,Z 476.03,A -85,B 0,C 180,E1 8638.013,E2 8638.013} C_VEL
LIN {X 0,Y 435.916,Z 476.03,A -85,B 0,C 180,E1 8643.986,E2 8643.986} C_VEL
LIN {X 0,Y 435.689,Z 476.03,A -85,B 0,C 180,E1 8650.009,E2 8650.009} C_VEL
LIN {X 0,Y 435.518,Z 476.03,A -85,B 0,C 180,E1 8656.15,E2 8656.15} C_VEL
LIN {X 0,Y 435.352,Z 476.03,A -85,B 0,C 180,E1 8662.495,E2 8662.495} C_VEL
LIN {X 0,Y 435.083,Z 476.03,A -85,B 0,C 180,E1 8669.158,E2 8669.158} C_VEL
LIN {X 0,Y 435.054,Z 476.03,A -85,B 0,C 180,E1 8673.839,E2 8673.839} C_VEL
LIN {X 0,Y 434.967,Z 476.03,A -85,B 0,C 180,E1 8680.021,E2 8680.021} C_VEL
LIN {X 0,Y 435.022,Z 476.03,A -85,B 0,C 180,E1 8685.885,E2 8685.885} C_VEL
LIN {X 0,Y 434.941,Z 476.03,A -85,B 0,C 180,E1 8691.2,E2 8691.2} C_VEL
LIN {X 0,Y 435.032,Z 476.03,A -85,B 0,C 180,E1 8698.529,E2 8698.529} C_VEL
LIN {X 0,Y 435.316,Z 476.03,A -85,B 0,C 180,E1 8705.608,E2 8705.608} C_VEL
LIN {X 0,Y 452.176,Z 513.798,A -85,B 0,C 180,E1 8708.808,E2 8708.808} C_VEL
LIN {X 0,Y 459.549,Z 536.589,A -85,B 0,C 180,E1 8710.824,E2 8710.824} C_VEL
LIN {X 0,Y 455.048,Z 573.349,A -85,B 0,C 180,E1 8713.323,E2 8713.323} C_VEL
LIN {X 0,Y 450.014,Z 606.594,A -85,B 0,C 180,E1 8716.502,E2 8716.502} C_VEL
LIN {X 0,Y 445.313,Z 635.323,A -85,B 0,C 180,E1 8720.212,E2 8720.212} C_VEL
LIN {X 0,Y 441.313,Z 660.527,A -85,B 0,C 180,E1 8724.586,E2 8724.586} C_VEL
LIN {X 0,Y 438.659,Z 679.524,A -85,B 0,C 180,E1 8729.011,E2 8729.011} C_VEL
LIN {X 0,Y 437.048,Z 694.702,A -85,B 0,C 180,E1 8733.973,E2 8733.973} C_VEL
LIN {X 0,Y 436.404,Z 705.203,A -85,B 0,C 180,E1 8738.969,E2 8738.969} C_VEL
LIN {X 0,Y 435.993,Z 710.257,A -85,B 0,C 180,E1 8743.501,E2 8743.501} C_VEL
LIN {X 0,Y 435.817,Z 711.257,A -85,B 0,C 180,E1 8748.221,E2 8748.221} C_VEL
LIN {X 0,Y 436.214,Z 707.356,A -85,B 0,C 180,E1 8753.432,E2 8753.432} C_VEL
LIN {X 0,Y 436.77,Z 698.832,A -85,B 0,C 180,E1 8758.233,E2 8758.233} C_VEL
LIN {X 0,Y 438.193,Z 684.184,A -85,B 0,C 180,E1 8763.564,E2 8763.564} C_VEL
LIN {X 0,Y 440.822,Z 664.148,A -85,B 0,C 180,E1 8768.598,E2 8768.598} C_VEL
LIN {X 0,Y 444.735,Z 639.174,A -85,B 0,C 180,E1 8773.122,E2 8773.122} C_VEL
LIN {X 0,Y 449.418,Z 610.273,A -85,B 0,C 180,E1 8776.992,E2 8776.992} C_VEL
LIN {X 0,Y 454.047,Z 579.2,A -85,B 0,C 180,E1 8780.084,E2 8780.084} C_VEL
LIN {X 0,Y 458.398,Z 544.412,A -85,B 0,C 180,E1 8782.603,E2 8782.603} C_VEL
LIN {X 0,Y 458.991,Z 534.7,A -85,B 0,C 180,E1 8783.196,E2 8783.196} C_VEL
LIN {X 0,Y 445.594,Z 498.65,A -85,B 0,C 180,E1 8786.41,E2 8786.41} C_VEL
LIN {X 0,Y 435.147,Z 476.03,A -85,B 0,C 180,E1 8788.419,E2 8788.419} C_VEL
LIN {X 0,Y 435.2,Z 476.03,A -85,B 0,C 180,E1 8795.322,E2 8795.322} C_VEL
LIN {X 0,Y 435.377,Z 476.03,A -85,B 0,C 180,E1 8796.658,E2 8796.658} C_VEL
LIN {X 0,Y 444.76,Z 511.699,A -85,B 0,C 180,E1 8797.939,E2 8797.939} C_VEL
LIN {X 0,Y 443.794,Z 543.664,A -85,B 0,C 180,E1 8799.425,E2 8799.425} C_VEL
LIN {X 0,Y 442.347,Z 571.808,A -85,B 0,C 180,E1 8801.54,E2 8801.54} C_VEL
LIN {X 0,Y 440.668,Z 597.386,A -85,B 0,C 180,E1 8804.377,E2 8804.377} C_VEL
LIN {X 0,Y 439.414,Z 617.18,A -85,B 0,C 180,E1 8807.561,E2 8807.561} C_VEL
LIN {X 0,Y 438.425,Z 632.073,A -85,B 0,C 180,E1 8811.057,E2 8811.057} C_VEL
LIN {X 0,Y 437.996,Z 642.53,A -85,B 0,C 180,E1 8815.039,E2 8815.039} C_VEL
LIN {X 0,Y 437.83,Z 646.546,A -85,B 0,C 180,E1 8818.015,E2 8818.015} C_VEL
LIN {X 0,Y 437.955,Z 647.166,A -85,B 0,C 180,E1 8821.978,E2 8821.978} C_VEL
LIN {X 0,Y 438.402,Z 642.304,A -85,B 0,C 180,E1 8825.944,E2 8825.944} C_VEL
LIN {X 0,Y 439.03,Z 633.112,A -85,B 0,C 180,E1 8829.425,E2 8829.425} C_VEL
LIN {X 0,Y 440.308,Z 618.188,A -85,B 0,C 180,E1 8832.912,E2 8832.912} C_VEL
LIN {X 0,Y 441.702,Z 598.183,A -85,B 0,C 180,E1 8836.045,E2 8836.045} C_VEL
LIN {X 0,Y 443.313,Z 573.329,A -85,B 0,C 180,E1 8838.67,E2 8838.67} C_VEL
LIN {X 0,Y 444.449,Z 544.752,A -85,B 0,C 180,E1 8840.664,E2 8840.664} C_VEL
LIN {X 0,Y 444.916,Z 514.602,A -85,B 0,C 180,E1 8841.921,E2 8841.921} C_VEL
LIN {X 0,Y 441.428,Z 495.462,A -85,B 0,C 180,E1 8842.547,E2 8842.547} C_VEL
LIN {X 0,Y 435.446,Z 476.03,A -85,B 0,C 180,E1 8843.339,E2 8843.339} C_VEL
LIN {X 0,Y 435.038,Z 476.03,A -85,B 0,C 180,E1 8849.528,E2 8849.528} C_VEL
LIN {X 0,Y 434.94,Z 476.03,A -85,B 0,C 180,E1 8856.278,E2 8856.278} C_VEL
LIN {X 0,Y 434.992,Z 476.03,A -85,B 0,C 180,E1 8863.032,E2 8863.032} C_VEL
LIN {X 0,Y 435.001,Z 476.612,A -85,B 0,C 180,E1 8866.597,E2 8866.597} C_VEL
LIN {X 0,Y 440.505,Z 487.058,A -85,B 0,C 180,E1 8867.545,E2 8867.545} C_VEL
LIN {X 0,Y 454.047,Z 513.723,A -85,B 0,C 180,E1 8869.788,E2 8869.788} C_VEL
LIN {X 0,Y 463.4,Z 537.596,A -85,B 0,C 180,E1 8871.477,E2 8871.477} C_VEL
LIN {X 0,Y 459.022,Z 582.934,A -85,B 0,C 180,E1 8873.243,E2 8873.243} C_VEL
LIN {X 0,Y 457.803,Z 594.786,A -85,B 0,C 180,E1 8873.864,E2 8873.864} C_VEL
LIN {X 0,Y 452.42,Z 610.645,A -85,B 0,C 180,E1 8874.542,E2 8874.542} C_VEL
LIN {X 0,Y 447.365,Z 624.127,A -85,B 0,C 180,E1 8875.231,E2 8875.231} C_VEL
LIN {X 0,Y 447.067,Z 625.988,A -85,B 0,C 180,E1 8875.366,E2 8875.366} C_VEL
LIN {X 0,Y 442.16,Z 662.667,A -85,B 0,C 180,E1 8878.519,E2 8878.519} C_VEL
LIN {X 0,Y 437.654,Z 694.755,A -85,B 0,C 180,E1 8882.228,E2 8882.228} C_VEL
LIN {X 0,Y 433.759,Z 723.12,A -85,B 0,C 180,E1 8886.605,E2 8886.605} C_VEL
LIN {X 0,Y 430.947,Z 746.721,A -85,B 0,C 180,E1 8891.566,E2 8891.566} C_VEL
LIN {X 0,Y 429.353,Z 762.681,A -85,B 0,C 180,E1 8896.229,E2 8896.229} C_VEL
LIN {X 0,Y 428.685,Z 773.408,A -85,B 0,C 180,E1 8900.812,E2 8900.812} C_VEL
LIN {X 0,Y 428.307,Z 779.929,A -85,B 0,C 180,E1 8905.945,E2 8905.945} C_VEL
LIN {X 0,Y 428.372,Z 781.5,A -85,B 0,C 180,E1 8910,E2 8910} C_VEL
LIN {X 0,Y 428.352,Z 779.929,A -85,B 0,C 180,E1 8914.054,E2 8914.054} C_VEL
LIN {X 0,Y 428.695,Z 773.377,A -85,B 0,C 180,E1 8919.205,E2 8919.205} C_VEL
LIN {X 0,Y 429.506,Z 761.22,A -85,B 0,C 180,E1 8924.286,E2 8924.286} C_VEL
LIN {X 0,Y 431.373,Z 742.601,A -85,B 0,C 180,E1 8929.478,E2 8929.478} C_VEL
LIN {X 0,Y 434.386,Z 719.217,A -85,B 0,C 180,E1 8934.177,E2 8934.177} C_VEL
LIN {X 0,Y 438.595,Z 690.069,A -85,B 0,C 180,E1 8938.528,E2 8938.528} C_VEL
LIN {X 0,Y 443.538,Z 656.032,A -85,B 0,C 180,E1 8942.307,E2 8942.307} C_VEL
LIN {X 0,Y 448.838,Z 617.697,A -85,B 0,C 180,E1 8945.431,E2 8945.431} C_VEL
LIN {X 0,Y 453.736,Z 577.866,A -85,B 0,C 180,E1 8947.727,E2 8947.727} C_VEL
LIN {X 0,Y 457.218,Z 539.678,A -85,B 0,C 180,E1 8949.251,E2 8949.251} C_VEL
LIN {X 0,Y 447.65,Z 516.619,A -85,B 0,C 180,E1 8950.986,E2 8950.986} C_VEL
LIN {X 0,Y 435.605,Z 492.42,A -85,B 0,C 180,E1 8952.945,E2 8952.945} C_VEL
LIN {X 0,Y 427.145,Z 476.835,A -85,B 0,C 180,E1 8954.292,E2 8954.292} C_VEL
LIN {X 0,Y 426.993,Z 476.03,A -85,B 0,C 180,E1 8958.129,E2 8958.129} C_VEL
LIN {X 0,Y 427.015,Z 476.03,A -85,B 0,C 180,E1 8964.64,E2 8964.64} C_VEL
LIN {X 0,Y 427.172,Z 476.03,A -85,B 0,C 180,E1 8970.255,E2 8970.255} C_VEL
LIN {X 0,Y 427.325,Z 476.03,A -85,B 0,C 180,E1 8977.108,E2 8977.108} C_VEL
LIN {X 0,Y 427.59,Z 476.03,A -85,B 0,C 180,E1 8983.548,E2 8983.548} C_VEL
LIN {X 0,Y 427.798,Z 476.03,A -85,B 0,C 180,E1 8989.811,E2 8989.811} C_VEL
LIN {X 0,Y 428.135,Z 476.03,A -85,B 0,C 180,E1 8995.947,E2 8995.947} C_VEL
LIN {X 0,Y 428.274,Z 476.03,A -85,B 0,C 180,E1 9002.029,E2 9002.029} C_VEL
LIN {X 0,Y 427.913,Z 476.03,A -85,B 0,C 180,E1 9008.139,E2 9008.139} C_VEL
LIN {X 0,Y 427.621,Z 476.03,A -85,B 0,C 180,E1 9014.353,E2 9014.353} C_VEL
LIN {X 0,Y 427.442,Z 476.03,A -85,B 0,C 180,E1 9020.748,E2 9020.748} C_VEL
